//     PlcTask Inputs/GVL_iXlinker.EtherCAT_Master_EPPxxxx.Beckhoff_EPP3xxx.Beckhoff_EPP3xxxEK1122.A_0012_EPP3314_0002_0016.TC_Inputs_Channel_1.Status/Limit_2 <-> TC Inputs Channel 1/Status/Limit 2
//     PlcTask Inputs/GVL_iXlinker.EtherCAT_Master_EPPxxxx.Beckhoff_EPP3xxx.Beckhoff_EPP3xxxEK1122.A_0012_EPP3314_0002_0016.TC_Inputs_Channel_2.Status/Limit_1 <-> TC Inputs Channel 2/Status/Limit 1
//     PlcTask Inputs/GVL_iXlinker.EtherCAT_Master_EPPxxxx.Beckhoff_EPP3xxx.Beckhoff_EPP3xxxEK1122.A_0012_EPP3314_0002_0016.TC_Inputs_Channel_2.Status/Limit_2 <-> TC Inputs Channel 2/Status/Limit 2
//     PlcTask Inputs/GVL_iXlinker.EtherCAT_Master_EPPxxxx.Beckhoff_EPP3xxx.Beckhoff_EPP3xxxEK1122.A_0012_EPP3314_0002_0016.TC_Inputs_Channel_3.Status/Limit_1 <-> TC Inputs Channel 3/Status/Limit 1
//     PlcTask Inputs/GVL_iXlinker.EtherCAT_Master_EPPxxxx.Beckhoff_EPP3xxx.Beckhoff_EPP3xxxEK1122.A_0012_EPP3314_0002_0016.TC_Inputs_Channel_3.Status/Limit_2 <-> TC Inputs Channel 3/Status/Limit 2
//     PlcTask Inputs/GVL_iXlinker.EtherCAT_Master_EPPxxxx.Beckhoff_EPP3xxx.Beckhoff_EPP3xxxEK1122.A_0012_EPP3314_0002_0016.TC_Inputs_Channel_4.Status/Limit_1 <-> TC Inputs Channel 4/Status/Limit 1
//     PlcTask Inputs/GVL_iXlinker.EtherCAT_Master_EPPxxxx.Beckhoff_EPP3xxx.Beckhoff_EPP3xxxEK1122.A_0012_EPP3314_0002_0016.TC_Inputs_Channel_4.Status/Limit_2 <-> TC Inputs Channel 4/Status/Limit 2
//     PlcTask Inputs/GVL_iXlinker.EtherCAT_Master_EPPxxxx.Beckhoff_EPP3xxx.Beckhoff_EPP3xxxEK1122.A_0012_EPP3314_0002_0016.TC_Inputs_Channel_1.Status/Error <-> TC Inputs Channel 1/Status/Error
//     PlcTask Inputs/GVL_iXlinker.EtherCAT_Master_EPPxxxx.Beckhoff_EPP3xxx.Beckhoff_EPP3xxxEK1122.A_0012_EPP3314_0002_0016.TC_Inputs_Channel_2.Status/Error <-> TC Inputs Channel 2/Status/Error
//     PlcTask Inputs/GVL_iXlinker.EtherCAT_Master_EPPxxxx.Beckhoff_EPP3xxx.Beckhoff_EPP3xxxEK1122.A_0012_EPP3314_0002_0016.TC_Inputs_Channel_3.Status/Error <-> TC Inputs Channel 3/Status/Error
//     PlcTask Inputs/GVL_iXlinker.EtherCAT_Master_EPPxxxx.Beckhoff_EPP3xxx.Beckhoff_EPP3xxxEK1122.A_0012_EPP3314_0002_0016.TC_Inputs_Channel_4.Status/Error <-> TC Inputs Channel 4/Status/Error
//     PlcTask Inputs/GVL_iXlinker.EtherCAT_Master_EPPxxxx.Beckhoff_EPP3xxx.Beckhoff_EPP3xxxEK1122.A_0012_EPP3314_0002_0016.TC_Inputs_Channel_1.Status/TxPDO_State <-> TC Inputs Channel 1/Status/TxPDO State
//     PlcTask Inputs/GVL_iXlinker.EtherCAT_Master_EPPxxxx.Beckhoff_EPP3xxx.Beckhoff_EPP3xxxEK1122.A_0012_EPP3314_0002_0016.TC_Inputs_Channel_2.Status/TxPDO_State <-> TC Inputs Channel 2/Status/TxPDO State
//     PlcTask Inputs/GVL_iXlinker.EtherCAT_Master_EPPxxxx.Beckhoff_EPP3xxx.Beckhoff_EPP3xxxEK1122.A_0012_EPP3314_0002_0016.TC_Inputs_Channel_3.Status/TxPDO_State <-> TC Inputs Channel 3/Status/TxPDO State
//     PlcTask Inputs/GVL_iXlinker.EtherCAT_Master_EPPxxxx.Beckhoff_EPP3xxx.Beckhoff_EPP3xxxEK1122.A_0012_EPP3314_0002_0016.TC_Inputs_Channel_4.Status/TxPDO_State <-> TC Inputs Channel 4/Status/TxPDO State
//     PlcTask Inputs/GVL_iXlinker.EtherCAT_Master_EPPxxxx.Beckhoff_EPP3xxx.Beckhoff_EPP3xxxEK1122.A_0012_EPP3314_0002_0016.TC_Inputs_Channel_1.Status/TxPDO_Toggle <-> TC Inputs Channel 1/Status/TxPDO Toggle
//     PlcTask Inputs/GVL_iXlinker.EtherCAT_Master_EPPxxxx.Beckhoff_EPP3xxx.Beckhoff_EPP3xxxEK1122.A_0012_EPP3314_0002_0016.TC_Inputs_Channel_2.Status/TxPDO_Toggle <-> TC Inputs Channel 2/Status/TxPDO Toggle
//     PlcTask Inputs/GVL_iXlinker.EtherCAT_Master_EPPxxxx.Beckhoff_EPP3xxx.Beckhoff_EPP3xxxEK1122.A_0012_EPP3314_0002_0016.TC_Inputs_Channel_3.Status/TxPDO_Toggle <-> TC Inputs Channel 3/Status/TxPDO Toggle
//     PlcTask Inputs/GVL_iXlinker.EtherCAT_Master_EPPxxxx.Beckhoff_EPP3xxx.Beckhoff_EPP3xxxEK1122.A_0012_EPP3314_0002_0016.TC_Inputs_Channel_4.Status/TxPDO_Toggle <-> TC Inputs Channel 4/Status/TxPDO Toggle
//     PlcTask Inputs/GVL_iXlinker.EtherCAT_Master_EPPxxxx.Beckhoff_EPP3xxx.Beckhoff_EPP3xxxEK1122.A_0012_EPP3314_0002_0016.TC_Inputs_Channel_1.Value <-> TC Inputs Channel 1/Value
//     PlcTask Inputs/GVL_iXlinker.EtherCAT_Master_EPPxxxx.Beckhoff_EPP3xxx.Beckhoff_EPP3xxxEK1122.A_0012_EPP3314_0002_0016.TC_Inputs_Channel_2.Value <-> TC Inputs Channel 2/Value
//     PlcTask Inputs/GVL_iXlinker.EtherCAT_Master_EPPxxxx.Beckhoff_EPP3xxx.Beckhoff_EPP3xxxEK1122.A_0012_EPP3314_0002_0016.TC_Inputs_Channel_3.Value <-> TC Inputs Channel 3/Value
//     PlcTask Inputs/GVL_iXlinker.EtherCAT_Master_EPPxxxx.Beckhoff_EPP3xxx.Beckhoff_EPP3xxxEK1122.A_0012_EPP3314_0002_0016.TC_Inputs_Channel_4.Value <-> TC Inputs Channel 4/Value
//     PlcTask Inputs/GVL_iXlinker.EtherCAT_Master_EPPxxxx.Beckhoff_EPP3xxx.Beckhoff_EPP3xxxEK1122.A_0012_EPP3314_0002_0016.WcState.WcState <-> WcState/WcState
//     PlcTask Inputs/GVL_iXlinker.EtherCAT_Master_EPPxxxx.Beckhoff_EPP3xxx.Beckhoff_EPP3xxxEK1122.A_0012_EPP3314_0002_0016.WcState.InputToggle <-> WcState/InputToggle
//     PlcTask Inputs/GVL_iXlinker.EtherCAT_Master_EPPxxxx.Beckhoff_EPP3xxx.Beckhoff_EPP3xxxEK1122.A_0012_EPP3314_0002_0016.InfoData.AdsAddr <-> InfoData/AdsAddr
//     PlcTask Inputs/GVL_iXlinker.EtherCAT_Master_EPPxxxx.Beckhoff_EPP3xxx.Beckhoff_EPP3xxxEK1122.A_0012_EPP3314_0002_0016.InfoData.State <-> InfoData/State
//   PLC/PLC Instance <-> EtherCAT Master EPPxxxx/Beckhoff EPP3xxx/Beckhoff EPP3xxxEK1122/A_0013(EPP3314-0002-0017)
//     PlcTask Inputs/GVL_iXlinker.EtherCAT_Master_EPPxxxx.Beckhoff_EPP3xxx.Beckhoff_EPP3xxxEK1122.A_0013_EPP3314_0002_0017.TC_Inputs_Channel_1.Status/Underrange <-> TC Inputs Channel 1/Status/Underrange
//     PlcTask Inputs/GVL_iXlinker.EtherCAT_Master_EPPxxxx.Beckhoff_EPP3xxx.Beckhoff_EPP3xxxEK1122.A_0013_EPP3314_0002_0017.TC_Inputs_Channel_2.Status/Underrange <-> TC Inputs Channel 2/Status/Underrange
//     PlcTask Inputs/GVL_iXlinker.EtherCAT_Master_EPPxxxx.Beckhoff_EPP3xxx.Beckhoff_EPP3xxxEK1122.A_0013_EPP3314_0002_0017.TC_Inputs_Channel_3.Status/Underrange <-> TC Inputs Channel 3/Status/Underrange
//     PlcTask Inputs/GVL_iXlinker.EtherCAT_Master_EPPxxxx.Beckhoff_EPP3xxx.Beckhoff_EPP3xxxEK1122.A_0013_EPP3314_0002_0017.TC_Inputs_Channel_4.Status/Underrange <-> TC Inputs Channel 4/Status/Underrange
//     PlcTask Inputs/GVL_iXlinker.EtherCAT_Master_EPPxxxx.Beckhoff_EPP3xxx.Beckhoff_EPP3xxxEK1122.A_0013_EPP3314_0002_0017.TC_Inputs_Channel_1.Status/Overrange <-> TC Inputs Channel 1/Status/Overrange
//     PlcTask Inputs/GVL_iXlinker.EtherCAT_Master_EPPxxxx.Beckhoff_EPP3xxx.Beckhoff_EPP3xxxEK1122.A_0013_EPP3314_0002_0017.TC_Inputs_Channel_2.Status/Overrange <-> TC Inputs Channel 2/Status/Overrange
//     PlcTask Inputs/GVL_iXlinker.EtherCAT_Master_EPPxxxx.Beckhoff_EPP3xxx.Beckhoff_EPP3xxxEK1122.A_0013_EPP3314_0002_0017.TC_Inputs_Channel_3.Status/Overrange <-> TC Inputs Channel 3/Status/Overrange
//     PlcTask Inputs/GVL_iXlinker.EtherCAT_Master_EPPxxxx.Beckhoff_EPP3xxx.Beckhoff_EPP3xxxEK1122.A_0013_EPP3314_0002_0017.TC_Inputs_Channel_4.Status/Overrange <-> TC Inputs Channel 4/Status/Overrange
//     PlcTask Inputs/GVL_iXlinker.EtherCAT_Master_EPPxxxx.Beckhoff_EPP3xxx.Beckhoff_EPP3xxxEK1122.A_0013_EPP3314_0002_0017.TC_Inputs_Channel_1.Status/Limit_1 <-> TC Inputs Channel 1/Status/Limit 1
//     PlcTask Inputs/GVL_iXlinker.EtherCAT_Master_EPPxxxx.Beckhoff_EPP3xxx.Beckhoff_EPP3xxxEK1122.A_0013_EPP3314_0002_0017.TC_Inputs_Channel_1.Status/Limit_2 <-> TC Inputs Channel 1/Status/Limit 2
//     PlcTask Inputs/GVL_iXlinker.EtherCAT_Master_EPPxxxx.Beckhoff_EPP3xxx.Beckhoff_EPP3xxxEK1122.A_0013_EPP3314_0002_0017.TC_Inputs_Channel_2.Status/Limit_1 <-> TC Inputs Channel 2/Status/Limit 1
//     PlcTask Inputs/GVL_iXlinker.EtherCAT_Master_EPPxxxx.Beckhoff_EPP3xxx.Beckhoff_EPP3xxxEK1122.A_0013_EPP3314_0002_0017.TC_Inputs_Channel_2.Status/Limit_2 <-> TC Inputs Channel 2/Status/Limit 2
//     PlcTask Inputs/GVL_iXlinker.EtherCAT_Master_EPPxxxx.Beckhoff_EPP3xxx.Beckhoff_EPP3xxxEK1122.A_0013_EPP3314_0002_0017.TC_Inputs_Channel_3.Status/Limit_1 <-> TC Inputs Channel 3/Status/Limit 1
//     PlcTask Inputs/GVL_iXlinker.EtherCAT_Master_EPPxxxx.Beckhoff_EPP3xxx.Beckhoff_EPP3xxxEK1122.A_0013_EPP3314_0002_0017.TC_Inputs_Channel_3.Status/Limit_2 <-> TC Inputs Channel 3/Status/Limit 2
//     PlcTask Inputs/GVL_iXlinker.EtherCAT_Master_EPPxxxx.Beckhoff_EPP3xxx.Beckhoff_EPP3xxxEK1122.A_0013_EPP3314_0002_0017.TC_Inputs_Channel_4.Status/Limit_1 <-> TC Inputs Channel 4/Status/Limit 1
//     PlcTask Inputs/GVL_iXlinker.EtherCAT_Master_EPPxxxx.Beckhoff_EPP3xxx.Beckhoff_EPP3xxxEK1122.A_0013_EPP3314_0002_0017.TC_Inputs_Channel_4.Status/Limit_2 <-> TC Inputs Channel 4/Status/Limit 2
//     PlcTask Inputs/GVL_iXlinker.EtherCAT_Master_EPPxxxx.Beckhoff_EPP3xxx.Beckhoff_EPP3xxxEK1122.A_0013_EPP3314_0002_0017.TC_Inputs_Channel_1.Status/Error <-> TC Inputs Channel 1/Status/Error
//     PlcTask Inputs/GVL_iXlinker.EtherCAT_Master_EPPxxxx.Beckhoff_EPP3xxx.Beckhoff_EPP3xxxEK1122.A_0013_EPP3314_0002_0017.TC_Inputs_Channel_2.Status/Error <-> TC Inputs Channel 2/Status/Error
//     PlcTask Inputs/GVL_iXlinker.EtherCAT_Master_EPPxxxx.Beckhoff_EPP3xxx.Beckhoff_EPP3xxxEK1122.A_0013_EPP3314_0002_0017.TC_Inputs_Channel_3.Status/Error <-> TC Inputs Channel 3/Status/Error
//     PlcTask Inputs/GVL_iXlinker.EtherCAT_Master_EPPxxxx.Beckhoff_EPP3xxx.Beckhoff_EPP3xxxEK1122.A_0013_EPP3314_0002_0017.TC_Inputs_Channel_4.Status/Error <-> TC Inputs Channel 4/Status/Error
//     PlcTask Inputs/GVL_iXlinker.EtherCAT_Master_EPPxxxx.Beckhoff_EPP3xxx.Beckhoff_EPP3xxxEK1122.A_0013_EPP3314_0002_0017.TC_Inputs_Channel_1.Status/TxPDO_State <-> TC Inputs Channel 1/Status/TxPDO State
//     PlcTask Inputs/GVL_iXlinker.EtherCAT_Master_EPPxxxx.Beckhoff_EPP3xxx.Beckhoff_EPP3xxxEK1122.A_0013_EPP3314_0002_0017.TC_Inputs_Channel_2.Status/TxPDO_State <-> TC Inputs Channel 2/Status/TxPDO State
//     PlcTask Inputs/GVL_iXlinker.EtherCAT_Master_EPPxxxx.Beckhoff_EPP3xxx.Beckhoff_EPP3xxxEK1122.A_0013_EPP3314_0002_0017.TC_Inputs_Channel_3.Status/TxPDO_State <-> TC Inputs Channel 3/Status/TxPDO State
//     PlcTask Inputs/GVL_iXlinker.EtherCAT_Master_EPPxxxx.Beckhoff_EPP3xxx.Beckhoff_EPP3xxxEK1122.A_0013_EPP3314_0002_0017.TC_Inputs_Channel_4.Status/TxPDO_State <-> TC Inputs Channel 4/Status/TxPDO State
//     PlcTask Inputs/GVL_iXlinker.EtherCAT_Master_EPPxxxx.Beckhoff_EPP3xxx.Beckhoff_EPP3xxxEK1122.A_0013_EPP3314_0002_0017.TC_Inputs_Channel_1.Status/TxPDO_Toggle <-> TC Inputs Channel 1/Status/TxPDO Toggle
//     PlcTask Inputs/GVL_iXlinker.EtherCAT_Master_EPPxxxx.Beckhoff_EPP3xxx.Beckhoff_EPP3xxxEK1122.A_0013_EPP3314_0002_0017.TC_Inputs_Channel_2.Status/TxPDO_Toggle <-> TC Inputs Channel 2/Status/TxPDO Toggle
//     PlcTask Inputs/GVL_iXlinker.EtherCAT_Master_EPPxxxx.Beckhoff_EPP3xxx.Beckhoff_EPP3xxxEK1122.A_0013_EPP3314_0002_0017.TC_Inputs_Channel_3.Status/TxPDO_Toggle <-> TC Inputs Channel 3/Status/TxPDO Toggle
//     PlcTask Inputs/GVL_iXlinker.EtherCAT_Master_EPPxxxx.Beckhoff_EPP3xxx.Beckhoff_EPP3xxxEK1122.A_0013_EPP3314_0002_0017.TC_Inputs_Channel_4.Status/TxPDO_Toggle <-> TC Inputs Channel 4/Status/TxPDO Toggle
//     PlcTask Inputs/GVL_iXlinker.EtherCAT_Master_EPPxxxx.Beckhoff_EPP3xxx.Beckhoff_EPP3xxxEK1122.A_0013_EPP3314_0002_0017.TC_Inputs_Channel_1.Value <-> TC Inputs Channel 1/Value
//     PlcTask Inputs/GVL_iXlinker.EtherCAT_Master_EPPxxxx.Beckhoff_EPP3xxx.Beckhoff_EPP3xxxEK1122.A_0013_EPP3314_0002_0017.TC_Inputs_Channel_2.Value <-> TC Inputs Channel 2/Value
//     PlcTask Inputs/GVL_iXlinker.EtherCAT_Master_EPPxxxx.Beckhoff_EPP3xxx.Beckhoff_EPP3xxxEK1122.A_0013_EPP3314_0002_0017.TC_Inputs_Channel_3.Value <-> TC Inputs Channel 3/Value
//     PlcTask Inputs/GVL_iXlinker.EtherCAT_Master_EPPxxxx.Beckhoff_EPP3xxx.Beckhoff_EPP3xxxEK1122.A_0013_EPP3314_0002_0017.TC_Inputs_Channel_4.Value <-> TC Inputs Channel 4/Value
//     PlcTask Inputs/GVL_iXlinker.EtherCAT_Master_EPPxxxx.Beckhoff_EPP3xxx.Beckhoff_EPP3xxxEK1122.A_0013_EPP3314_0002_0017.WcState.WcState <-> WcState/WcState
//     PlcTask Inputs/GVL_iXlinker.EtherCAT_Master_EPPxxxx.Beckhoff_EPP3xxx.Beckhoff_EPP3xxxEK1122.A_0013_EPP3314_0002_0017.WcState.InputToggle <-> WcState/InputToggle
//     PlcTask Inputs/GVL_iXlinker.EtherCAT_Master_EPPxxxx.Beckhoff_EPP3xxx.Beckhoff_EPP3xxxEK1122.A_0013_EPP3314_0002_0017.InfoData.AdsAddr <-> InfoData/AdsAddr
//     PlcTask Inputs/GVL_iXlinker.EtherCAT_Master_EPPxxxx.Beckhoff_EPP3xxx.Beckhoff_EPP3xxxEK1122.A_0013_EPP3314_0002_0017.InfoData.State <-> InfoData/State
//   PLC/PLC Instance <-> EtherCAT Master EPPxxxx/Beckhoff EPP3xxx/Beckhoff EPP3xxxEK1122/A_0014(EPP3314-0002-0018)
//     PlcTask Inputs/GVL_iXlinker.EtherCAT_Master_EPPxxxx.Beckhoff_EPP3xxx.Beckhoff_EPP3xxxEK1122.A_0014_EPP3314_0002_0018.TC_Inputs_Channel_1.Status/Underrange <-> TC Inputs Channel 1/Status/Underrange
//     PlcTask Inputs/GVL_iXlinker.EtherCAT_Master_EPPxxxx.Beckhoff_EPP3xxx.Beckhoff_EPP3xxxEK1122.A_0014_EPP3314_0002_0018.TC_Inputs_Channel_2.Status/Underrange <-> TC Inputs Channel 2/Status/Underrange
//     PlcTask Inputs/GVL_iXlinker.EtherCAT_Master_EPPxxxx.Beckhoff_EPP3xxx.Beckhoff_EPP3xxxEK1122.A_0014_EPP3314_0002_0018.TC_Inputs_Channel_3.Status/Underrange <-> TC Inputs Channel 3/Status/Underrange
//     PlcTask Inputs/GVL_iXlinker.EtherCAT_Master_EPPxxxx.Beckhoff_EPP3xxx.Beckhoff_EPP3xxxEK1122.A_0014_EPP3314_0002_0018.TC_Inputs_Channel_4.Status/Underrange <-> TC Inputs Channel 4/Status/Underrange
//     PlcTask Inputs/GVL_iXlinker.EtherCAT_Master_EPPxxxx.Beckhoff_EPP3xxx.Beckhoff_EPP3xxxEK1122.A_0014_EPP3314_0002_0018.TC_Inputs_Channel_1.Status/Overrange <-> TC Inputs Channel 1/Status/Overrange
//     PlcTask Inputs/GVL_iXlinker.EtherCAT_Master_EPPxxxx.Beckhoff_EPP3xxx.Beckhoff_EPP3xxxEK1122.A_0014_EPP3314_0002_0018.TC_Inputs_Channel_2.Status/Overrange <-> TC Inputs Channel 2/Status/Overrange
//     PlcTask Inputs/GVL_iXlinker.EtherCAT_Master_EPPxxxx.Beckhoff_EPP3xxx.Beckhoff_EPP3xxxEK1122.A_0014_EPP3314_0002_0018.TC_Inputs_Channel_3.Status/Overrange <-> TC Inputs Channel 3/Status/Overrange
//     PlcTask Inputs/GVL_iXlinker.EtherCAT_Master_EPPxxxx.Beckhoff_EPP3xxx.Beckhoff_EPP3xxxEK1122.A_0014_EPP3314_0002_0018.TC_Inputs_Channel_4.Status/Overrange <-> TC Inputs Channel 4/Status/Overrange
//     PlcTask Inputs/GVL_iXlinker.EtherCAT_Master_EPPxxxx.Beckhoff_EPP3xxx.Beckhoff_EPP3xxxEK1122.A_0014_EPP3314_0002_0018.TC_Inputs_Channel_1.Status/Limit_1 <-> TC Inputs Channel 1/Status/Limit 1
//     PlcTask Inputs/GVL_iXlinker.EtherCAT_Master_EPPxxxx.Beckhoff_EPP3xxx.Beckhoff_EPP3xxxEK1122.A_0014_EPP3314_0002_0018.TC_Inputs_Channel_1.Status/Limit_2 <-> TC Inputs Channel 1/Status/Limit 2
//     PlcTask Inputs/GVL_iXlinker.EtherCAT_Master_EPPxxxx.Beckhoff_EPP3xxx.Beckhoff_EPP3xxxEK1122.A_0014_EPP3314_0002_0018.TC_Inputs_Channel_2.Status/Limit_1 <-> TC Inputs Channel 2/Status/Limit 1
//     PlcTask Inputs/GVL_iXlinker.EtherCAT_Master_EPPxxxx.Beckhoff_EPP3xxx.Beckhoff_EPP3xxxEK1122.A_0014_EPP3314_0002_0018.TC_Inputs_Channel_2.Status/Limit_2 <-> TC Inputs Channel 2/Status/Limit 2
//     PlcTask Inputs/GVL_iXlinker.EtherCAT_Master_EPPxxxx.Beckhoff_EPP3xxx.Beckhoff_EPP3xxxEK1122.A_0014_EPP3314_0002_0018.TC_Inputs_Channel_3.Status/Limit_1 <-> TC Inputs Channel 3/Status/Limit 1
//     PlcTask Inputs/GVL_iXlinker.EtherCAT_Master_EPPxxxx.Beckhoff_EPP3xxx.Beckhoff_EPP3xxxEK1122.A_0014_EPP3314_0002_0018.TC_Inputs_Channel_3.Status/Limit_2 <-> TC Inputs Channel 3/Status/Limit 2
//     PlcTask Inputs/GVL_iXlinker.EtherCAT_Master_EPPxxxx.Beckhoff_EPP3xxx.Beckhoff_EPP3xxxEK1122.A_0014_EPP3314_0002_0018.TC_Inputs_Channel_4.Status/Limit_1 <-> TC Inputs Channel 4/Status/Limit 1
//     PlcTask Inputs/GVL_iXlinker.EtherCAT_Master_EPPxxxx.Beckhoff_EPP3xxx.Beckhoff_EPP3xxxEK1122.A_0014_EPP3314_0002_0018.TC_Inputs_Channel_4.Status/Limit_2 <-> TC Inputs Channel 4/Status/Limit 2
//     PlcTask Inputs/GVL_iXlinker.EtherCAT_Master_EPPxxxx.Beckhoff_EPP3xxx.Beckhoff_EPP3xxxEK1122.A_0014_EPP3314_0002_0018.TC_Inputs_Channel_1.Status/Error <-> TC Inputs Channel 1/Status/Error
//     PlcTask Inputs/GVL_iXlinker.EtherCAT_Master_EPPxxxx.Beckhoff_EPP3xxx.Beckhoff_EPP3xxxEK1122.A_0014_EPP3314_0002_0018.TC_Inputs_Channel_2.Status/Error <-> TC Inputs Channel 2/Status/Error
//     PlcTask Inputs/GVL_iXlinker.EtherCAT_Master_EPPxxxx.Beckhoff_EPP3xxx.Beckhoff_EPP3xxxEK1122.A_0014_EPP3314_0002_0018.TC_Inputs_Channel_3.Status/Error <-> TC Inputs Channel 3/Status/Error
//     PlcTask Inputs/GVL_iXlinker.EtherCAT_Master_EPPxxxx.Beckhoff_EPP3xxx.Beckhoff_EPP3xxxEK1122.A_0014_EPP3314_0002_0018.TC_Inputs_Channel_4.Status/Error <-> TC Inputs Channel 4/Status/Error
//     PlcTask Inputs/GVL_iXlinker.EtherCAT_Master_EPPxxxx.Beckhoff_EPP3xxx.Beckhoff_EPP3xxxEK1122.A_0014_EPP3314_0002_0018.TC_Inputs_Channel_1.Status/TxPDO_State <-> TC Inputs Channel 1/Status/TxPDO State
//     PlcTask Inputs/GVL_iXlinker.EtherCAT_Master_EPPxxxx.Beckhoff_EPP3xxx.Beckhoff_EPP3xxxEK1122.A_0014_EPP3314_0002_0018.TC_Inputs_Channel_2.Status/TxPDO_State <-> TC Inputs Channel 2/Status/TxPDO State
//     PlcTask Inputs/GVL_iXlinker.EtherCAT_Master_EPPxxxx.Beckhoff_EPP3xxx.Beckhoff_EPP3xxxEK1122.A_0014_EPP3314_0002_0018.TC_Inputs_Channel_3.Status/TxPDO_State <-> TC Inputs Channel 3/Status/TxPDO State
//     PlcTask Inputs/GVL_iXlinker.EtherCAT_Master_EPPxxxx.Beckhoff_EPP3xxx.Beckhoff_EPP3xxxEK1122.A_0014_EPP3314_0002_0018.TC_Inputs_Channel_4.Status/TxPDO_State <-> TC Inputs Channel 4/Status/TxPDO State
//     PlcTask Inputs/GVL_iXlinker.EtherCAT_Master_EPPxxxx.Beckhoff_EPP3xxx.Beckhoff_EPP3xxxEK1122.A_0014_EPP3314_0002_0018.TC_Inputs_Channel_1.Status/TxPDO_Toggle <-> TC Inputs Channel 1/Status/TxPDO Toggle
//     PlcTask Inputs/GVL_iXlinker.EtherCAT_Master_EPPxxxx.Beckhoff_EPP3xxx.Beckhoff_EPP3xxxEK1122.A_0014_EPP3314_0002_0018.TC_Inputs_Channel_2.Status/TxPDO_Toggle <-> TC Inputs Channel 2/Status/TxPDO Toggle
//     PlcTask Inputs/GVL_iXlinker.EtherCAT_Master_EPPxxxx.Beckhoff_EPP3xxx.Beckhoff_EPP3xxxEK1122.A_0014_EPP3314_0002_0018.TC_Inputs_Channel_3.Status/TxPDO_Toggle <-> TC Inputs Channel 3/Status/TxPDO Toggle
//     PlcTask Inputs/GVL_iXlinker.EtherCAT_Master_EPPxxxx.Beckhoff_EPP3xxx.Beckhoff_EPP3xxxEK1122.A_0014_EPP3314_0002_0018.TC_Inputs_Channel_4.Status/TxPDO_Toggle <-> TC Inputs Channel 4/Status/TxPDO Toggle
//     PlcTask Inputs/GVL_iXlinker.EtherCAT_Master_EPPxxxx.Beckhoff_EPP3xxx.Beckhoff_EPP3xxxEK1122.A_0014_EPP3314_0002_0018.TC_Inputs_Channel_1.Value <-> TC Inputs Channel 1/Value
//     PlcTask Inputs/GVL_iXlinker.EtherCAT_Master_EPPxxxx.Beckhoff_EPP3xxx.Beckhoff_EPP3xxxEK1122.A_0014_EPP3314_0002_0018.TC_Inputs_Channel_2.Value <-> TC Inputs Channel 2/Value
//     PlcTask Inputs/GVL_iXlinker.EtherCAT_Master_EPPxxxx.Beckhoff_EPP3xxx.Beckhoff_EPP3xxxEK1122.A_0014_EPP3314_0002_0018.TC_Inputs_Channel_3.Value <-> TC Inputs Channel 3/Value
//     PlcTask Inputs/GVL_iXlinker.EtherCAT_Master_EPPxxxx.Beckhoff_EPP3xxx.Beckhoff_EPP3xxxEK1122.A_0014_EPP3314_0002_0018.TC_Inputs_Channel_4.Value <-> TC Inputs Channel 4/Value
//     PlcTask Inputs/GVL_iXlinker.EtherCAT_Master_EPPxxxx.Beckhoff_EPP3xxx.Beckhoff_EPP3xxxEK1122.A_0014_EPP3314_0002_0018.WcState.WcState <-> WcState/WcState
//     PlcTask Inputs/GVL_iXlinker.EtherCAT_Master_EPPxxxx.Beckhoff_EPP3xxx.Beckhoff_EPP3xxxEK1122.A_0014_EPP3314_0002_0018.WcState.InputToggle <-> WcState/InputToggle
//     PlcTask Inputs/GVL_iXlinker.EtherCAT_Master_EPPxxxx.Beckhoff_EPP3xxx.Beckhoff_EPP3xxxEK1122.A_0014_EPP3314_0002_0018.InfoData.AdsAddr <-> InfoData/AdsAddr
//     PlcTask Inputs/GVL_iXlinker.EtherCAT_Master_EPPxxxx.Beckhoff_EPP3xxx.Beckhoff_EPP3xxxEK1122.A_0014_EPP3314_0002_0018.InfoData.State <-> InfoData/State
//   PLC/PLC Instance <-> EtherCAT Master EPPxxxx/Beckhoff EPP3xxx/Beckhoff EPP3xxxEK1122/A_0015(EPP3632-0001-0016)
//     PlcTask Inputs/GVL_iXlinker.EtherCAT_Master_EPPxxxx.Beckhoff_EPP3xxx.Beckhoff_EPP3xxxEK1122.A_0015_EPP3632_0001_0016.Ch1_Status.STATUS/Underrange <-> Ch1 Status/STATUS/Underrange
//     PlcTask Inputs/GVL_iXlinker.EtherCAT_Master_EPPxxxx.Beckhoff_EPP3xxx.Beckhoff_EPP3xxxEK1122.A_0015_EPP3632_0001_0016.Ch2_Status.STATUS/Underrange <-> Ch2 Status/STATUS/Underrange
//     PlcTask Inputs/GVL_iXlinker.EtherCAT_Master_EPPxxxx.Beckhoff_EPP3xxx.Beckhoff_EPP3xxxEK1122.A_0015_EPP3632_0001_0016.Ch1_Status.STATUS/Overrange <-> Ch1 Status/STATUS/Overrange
//     PlcTask Inputs/GVL_iXlinker.EtherCAT_Master_EPPxxxx.Beckhoff_EPP3xxx.Beckhoff_EPP3xxxEK1122.A_0015_EPP3632_0001_0016.Ch2_Status.STATUS/Overrange <-> Ch2 Status/STATUS/Overrange
//     PlcTask Inputs/GVL_iXlinker.EtherCAT_Master_EPPxxxx.Beckhoff_EPP3xxx.Beckhoff_EPP3xxxEK1122.A_0015_EPP3632_0001_0016.Ch1_Status.STATUS/Limit_1 <-> Ch1 Status/STATUS/Limit 1
//     PlcTask Inputs/GVL_iXlinker.EtherCAT_Master_EPPxxxx.Beckhoff_EPP3xxx.Beckhoff_EPP3xxxEK1122.A_0015_EPP3632_0001_0016.Ch1_Status.STATUS/Limit_2 <-> Ch1 Status/STATUS/Limit 2
//     PlcTask Inputs/GVL_iXlinker.EtherCAT_Master_EPPxxxx.Beckhoff_EPP3xxx.Beckhoff_EPP3xxxEK1122.A_0015_EPP3632_0001_0016.Ch2_Status.STATUS/Limit_1 <-> Ch2 Status/STATUS/Limit 1
//     PlcTask Inputs/GVL_iXlinker.EtherCAT_Master_EPPxxxx.Beckhoff_EPP3xxx.Beckhoff_EPP3xxxEK1122.A_0015_EPP3632_0001_0016.Ch2_Status.STATUS/Limit_2 <-> Ch2 Status/STATUS/Limit 2
//     PlcTask Inputs/GVL_iXlinker.EtherCAT_Master_EPPxxxx.Beckhoff_EPP3xxx.Beckhoff_EPP3xxxEK1122.A_0015_EPP3632_0001_0016.Ch1_Status.STATUS/Error <-> Ch1 Status/STATUS/Error
//     PlcTask Inputs/GVL_iXlinker.EtherCAT_Master_EPPxxxx.Beckhoff_EPP3xxx.Beckhoff_EPP3xxxEK1122.A_0015_EPP3632_0001_0016.Ch2_Status.STATUS/Error <-> Ch2 Status/STATUS/Error
//     PlcTask Inputs/GVL_iXlinker.EtherCAT_Master_EPPxxxx.Beckhoff_EPP3xxx.Beckhoff_EPP3xxxEK1122.A_0015_EPP3632_0001_0016.Ch1_Status.STATUS/Sync_error <-> Ch1 Status/STATUS/Sync error
//     PlcTask Inputs/GVL_iXlinker.EtherCAT_Master_EPPxxxx.Beckhoff_EPP3xxx.Beckhoff_EPP3xxxEK1122.A_0015_EPP3632_0001_0016.Ch2_Status.STATUS/Sync_error <-> Ch2 Status/STATUS/Sync error
//     PlcTask Inputs/GVL_iXlinker.EtherCAT_Master_EPPxxxx.Beckhoff_EPP3xxx.Beckhoff_EPP3xxxEK1122.A_0015_EPP3632_0001_0016.Ch1_Status.STATUS/TxPDO_State <-> Ch1 Status/STATUS/TxPDO State
//     PlcTask Inputs/GVL_iXlinker.EtherCAT_Master_EPPxxxx.Beckhoff_EPP3xxx.Beckhoff_EPP3xxxEK1122.A_0015_EPP3632_0001_0016.Ch2_Status.STATUS/TxPDO_State <-> Ch2 Status/STATUS/TxPDO State
//     PlcTask Inputs/GVL_iXlinker.EtherCAT_Master_EPPxxxx.Beckhoff_EPP3xxx.Beckhoff_EPP3xxxEK1122.A_0015_EPP3632_0001_0016.Ch1_Status.STATUS/TxPDO_Toggle <-> Ch1 Status/STATUS/TxPDO Toggle
//     PlcTask Inputs/GVL_iXlinker.EtherCAT_Master_EPPxxxx.Beckhoff_EPP3xxx.Beckhoff_EPP3xxxEK1122.A_0015_EPP3632_0001_0016.Ch2_Status.STATUS/TxPDO_Toggle <-> Ch2 Status/STATUS/TxPDO Toggle
//     PlcTask Inputs/GVL_iXlinker.EtherCAT_Master_EPPxxxx.Beckhoff_EPP3xxx.Beckhoff_EPP3xxxEK1122.A_0015_EPP3632_0001_0016.Ch1_Sample_0.Ch1_Value <-> Ch1 Sample 0/Ch1 Value
//     PlcTask Inputs/GVL_iXlinker.EtherCAT_Master_EPPxxxx.Beckhoff_EPP3xxx.Beckhoff_EPP3xxxEK1122.A_0015_EPP3632_0001_0016.Ch1_Sample_1.Ch1_Value <-> Ch1 Sample 1/Ch1 Value
//     PlcTask Inputs/GVL_iXlinker.EtherCAT_Master_EPPxxxx.Beckhoff_EPP3xxx.Beckhoff_EPP3xxxEK1122.A_0015_EPP3632_0001_0016.Ch1_Sample_2.Ch1_Value <-> Ch1 Sample 2/Ch1 Value
//     PlcTask Inputs/GVL_iXlinker.EtherCAT_Master_EPPxxxx.Beckhoff_EPP3xxx.Beckhoff_EPP3xxxEK1122.A_0015_EPP3632_0001_0016.Ch1_Sample_3.Ch1_Value <-> Ch1 Sample 3/Ch1 Value
//     PlcTask Inputs/GVL_iXlinker.EtherCAT_Master_EPPxxxx.Beckhoff_EPP3xxx.Beckhoff_EPP3xxxEK1122.A_0015_EPP3632_0001_0016.Ch1_Sample_4.Ch1_Value <-> Ch1 Sample 4/Ch1 Value
//     PlcTask Inputs/GVL_iXlinker.EtherCAT_Master_EPPxxxx.Beckhoff_EPP3xxx.Beckhoff_EPP3xxxEK1122.A_0015_EPP3632_0001_0016.Ch1_Sample_5.Ch1_Value <-> Ch1 Sample 5/Ch1 Value
//     PlcTask Inputs/GVL_iXlinker.EtherCAT_Master_EPPxxxx.Beckhoff_EPP3xxx.Beckhoff_EPP3xxxEK1122.A_0015_EPP3632_0001_0016.Ch1_Sample_6.Ch1_Value <-> Ch1 Sample 6/Ch1 Value
//     PlcTask Inputs/GVL_iXlinker.EtherCAT_Master_EPPxxxx.Beckhoff_EPP3xxx.Beckhoff_EPP3xxxEK1122.A_0015_EPP3632_0001_0016.Ch1_Sample_7.Ch1_Value <-> Ch1 Sample 7/Ch1 Value
//     PlcTask Inputs/GVL_iXlinker.EtherCAT_Master_EPPxxxx.Beckhoff_EPP3xxx.Beckhoff_EPP3xxxEK1122.A_0015_EPP3632_0001_0016.Ch1_Sample_8.Ch1_Value <-> Ch1 Sample 8/Ch1 Value
//     PlcTask Inputs/GVL_iXlinker.EtherCAT_Master_EPPxxxx.Beckhoff_EPP3xxx.Beckhoff_EPP3xxxEK1122.A_0015_EPP3632_0001_0016.Ch1_Sample_9.Ch1_Value <-> Ch1 Sample 9/Ch1 Value
//     PlcTask Inputs/GVL_iXlinker.EtherCAT_Master_EPPxxxx.Beckhoff_EPP3xxx.Beckhoff_EPP3xxxEK1122.A_0015_EPP3632_0001_0016.Ch2_Sample_0.Ch2_Value <-> Ch2 Sample 0/Ch2 Value
//     PlcTask Inputs/GVL_iXlinker.EtherCAT_Master_EPPxxxx.Beckhoff_EPP3xxx.Beckhoff_EPP3xxxEK1122.A_0015_EPP3632_0001_0016.Ch2_Sample_1.Ch2_Value <-> Ch2 Sample 1/Ch2 Value
//     PlcTask Inputs/GVL_iXlinker.EtherCAT_Master_EPPxxxx.Beckhoff_EPP3xxx.Beckhoff_EPP3xxxEK1122.A_0015_EPP3632_0001_0016.Ch2_Sample_2.Ch2_Value <-> Ch2 Sample 2/Ch2 Value
//     PlcTask Inputs/GVL_iXlinker.EtherCAT_Master_EPPxxxx.Beckhoff_EPP3xxx.Beckhoff_EPP3xxxEK1122.A_0015_EPP3632_0001_0016.Ch2_Sample_3.Ch2_Value <-> Ch2 Sample 3/Ch2 Value
//     PlcTask Inputs/GVL_iXlinker.EtherCAT_Master_EPPxxxx.Beckhoff_EPP3xxx.Beckhoff_EPP3xxxEK1122.A_0015_EPP3632_0001_0016.Ch2_Sample_4.Ch2_Value <-> Ch2 Sample 4/Ch2 Value
//     PlcTask Inputs/GVL_iXlinker.EtherCAT_Master_EPPxxxx.Beckhoff_EPP3xxx.Beckhoff_EPP3xxxEK1122.A_0015_EPP3632_0001_0016.Ch2_Sample_5.Ch2_Value <-> Ch2 Sample 5/Ch2 Value
//     PlcTask Inputs/GVL_iXlinker.EtherCAT_Master_EPPxxxx.Beckhoff_EPP3xxx.Beckhoff_EPP3xxxEK1122.A_0015_EPP3632_0001_0016.Ch2_Sample_6.Ch2_Value <-> Ch2 Sample 6/Ch2 Value
//     PlcTask Inputs/GVL_iXlinker.EtherCAT_Master_EPPxxxx.Beckhoff_EPP3xxx.Beckhoff_EPP3xxxEK1122.A_0015_EPP3632_0001_0016.Ch2_Sample_7.Ch2_Value <-> Ch2 Sample 7/Ch2 Value
//     PlcTask Inputs/GVL_iXlinker.EtherCAT_Master_EPPxxxx.Beckhoff_EPP3xxx.Beckhoff_EPP3xxxEK1122.A_0015_EPP3632_0001_0016.Ch2_Sample_8.Ch2_Value <-> Ch2 Sample 8/Ch2 Value
//     PlcTask Inputs/GVL_iXlinker.EtherCAT_Master_EPPxxxx.Beckhoff_EPP3xxx.Beckhoff_EPP3xxxEK1122.A_0015_EPP3632_0001_0016.Ch2_Sample_9.Ch2_Value <-> Ch2 Sample 9/Ch2 Value
//     PlcTask Inputs/GVL_iXlinker.EtherCAT_Master_EPPxxxx.Beckhoff_EPP3xxx.Beckhoff_EPP3xxxEK1122.A_0015_EPP3632_0001_0016.NextSync1Time.StartTimeNextLatch <-> NextSync1Time/StartTimeNextLatch
//     PlcTask Inputs/GVL_iXlinker.EtherCAT_Master_EPPxxxx.Beckhoff_EPP3xxx.Beckhoff_EPP3xxxEK1122.A_0015_EPP3632_0001_0016.Sample_Count.Sample_Count <-> Sample Count/Sample Count
//     PlcTask Inputs/GVL_iXlinker.EtherCAT_Master_EPPxxxx.Beckhoff_EPP3xxx.Beckhoff_EPP3xxxEK1122.A_0015_EPP3632_0001_0016.WcState.WcState <-> WcState/WcState
//     PlcTask Inputs/GVL_iXlinker.EtherCAT_Master_EPPxxxx.Beckhoff_EPP3xxx.Beckhoff_EPP3xxxEK1122.A_0015_EPP3632_0001_0016.WcState.InputToggle <-> WcState/InputToggle
//     PlcTask Inputs/GVL_iXlinker.EtherCAT_Master_EPPxxxx.Beckhoff_EPP3xxx.Beckhoff_EPP3xxxEK1122.A_0015_EPP3632_0001_0016.InfoData.AdsAddr <-> InfoData/AdsAddr
//     PlcTask Inputs/GVL_iXlinker.EtherCAT_Master_EPPxxxx.Beckhoff_EPP3xxx.Beckhoff_EPP3xxxEK1122.A_0015_EPP3632_0001_0016.InfoData.DcOutputShift <-> InfoData/DcOutputShift
//     PlcTask Inputs/GVL_iXlinker.EtherCAT_Master_EPPxxxx.Beckhoff_EPP3xxx.Beckhoff_EPP3xxxEK1122.A_0015_EPP3632_0001_0016.InfoData.DcInputShift <-> InfoData/DcInputShift
//     PlcTask Inputs/GVL_iXlinker.EtherCAT_Master_EPPxxxx.Beckhoff_EPP3xxx.Beckhoff_EPP3xxxEK1122.A_0015_EPP3632_0001_0016.InfoData.State <-> InfoData/State
//   PLC/PLC Instance <-> EtherCAT Master EPPxxxx/Beckhoff EPP3xxx/Beckhoff EPP3xxxEK1122/A_0016(EPP3632-0001-0017)
//     PlcTask Inputs/GVL_iXlinker.EtherCAT_Master_EPPxxxx.Beckhoff_EPP3xxx.Beckhoff_EPP3xxxEK1122.A_0016_EPP3632_0001_0017.Ch1_Status.STATUS/Underrange <-> Ch1 Status/STATUS/Underrange
//     PlcTask Inputs/GVL_iXlinker.EtherCAT_Master_EPPxxxx.Beckhoff_EPP3xxx.Beckhoff_EPP3xxxEK1122.A_0016_EPP3632_0001_0017.Ch2_Status.STATUS/Underrange <-> Ch2 Status/STATUS/Underrange
//     PlcTask Inputs/GVL_iXlinker.EtherCAT_Master_EPPxxxx.Beckhoff_EPP3xxx.Beckhoff_EPP3xxxEK1122.A_0016_EPP3632_0001_0017.Ch1_Status.STATUS/Overrange <-> Ch1 Status/STATUS/Overrange
//     PlcTask Inputs/GVL_iXlinker.EtherCAT_Master_EPPxxxx.Beckhoff_EPP3xxx.Beckhoff_EPP3xxxEK1122.A_0016_EPP3632_0001_0017.Ch2_Status.STATUS/Overrange <-> Ch2 Status/STATUS/Overrange
//     PlcTask Inputs/GVL_iXlinker.EtherCAT_Master_EPPxxxx.Beckhoff_EPP3xxx.Beckhoff_EPP3xxxEK1122.A_0016_EPP3632_0001_0017.Ch1_Status.STATUS/Limit_1 <-> Ch1 Status/STATUS/Limit 1
//     PlcTask Inputs/GVL_iXlinker.EtherCAT_Master_EPPxxxx.Beckhoff_EPP3xxx.Beckhoff_EPP3xxxEK1122.A_0016_EPP3632_0001_0017.Ch1_Status.STATUS/Limit_2 <-> Ch1 Status/STATUS/Limit 2
//     PlcTask Inputs/GVL_iXlinker.EtherCAT_Master_EPPxxxx.Beckhoff_EPP3xxx.Beckhoff_EPP3xxxEK1122.A_0016_EPP3632_0001_0017.Ch2_Status.STATUS/Limit_1 <-> Ch2 Status/STATUS/Limit 1
//     PlcTask Inputs/GVL_iXlinker.EtherCAT_Master_EPPxxxx.Beckhoff_EPP3xxx.Beckhoff_EPP3xxxEK1122.A_0016_EPP3632_0001_0017.Ch2_Status.STATUS/Limit_2 <-> Ch2 Status/STATUS/Limit 2
//     PlcTask Inputs/GVL_iXlinker.EtherCAT_Master_EPPxxxx.Beckhoff_EPP3xxx.Beckhoff_EPP3xxxEK1122.A_0016_EPP3632_0001_0017.Ch1_Status.STATUS/Error <-> Ch1 Status/STATUS/Error
//     PlcTask Inputs/GVL_iXlinker.EtherCAT_Master_EPPxxxx.Beckhoff_EPP3xxx.Beckhoff_EPP3xxxEK1122.A_0016_EPP3632_0001_0017.Ch2_Status.STATUS/Error <-> Ch2 Status/STATUS/Error
//     PlcTask Inputs/GVL_iXlinker.EtherCAT_Master_EPPxxxx.Beckhoff_EPP3xxx.Beckhoff_EPP3xxxEK1122.A_0016_EPP3632_0001_0017.Ch1_Status.STATUS/Sync_error <-> Ch1 Status/STATUS/Sync error
//     PlcTask Inputs/GVL_iXlinker.EtherCAT_Master_EPPxxxx.Beckhoff_EPP3xxx.Beckhoff_EPP3xxxEK1122.A_0016_EPP3632_0001_0017.Ch2_Status.STATUS/Sync_error <-> Ch2 Status/STATUS/Sync error
//     PlcTask Inputs/GVL_iXlinker.EtherCAT_Master_EPPxxxx.Beckhoff_EPP3xxx.Beckhoff_EPP3xxxEK1122.A_0016_EPP3632_0001_0017.Ch1_Status.STATUS/TxPDO_State <-> Ch1 Status/STATUS/TxPDO State
//     PlcTask Inputs/GVL_iXlinker.EtherCAT_Master_EPPxxxx.Beckhoff_EPP3xxx.Beckhoff_EPP3xxxEK1122.A_0016_EPP3632_0001_0017.Ch2_Status.STATUS/TxPDO_State <-> Ch2 Status/STATUS/TxPDO State
//     PlcTask Inputs/GVL_iXlinker.EtherCAT_Master_EPPxxxx.Beckhoff_EPP3xxx.Beckhoff_EPP3xxxEK1122.A_0016_EPP3632_0001_0017.Ch1_Status.STATUS/TxPDO_Toggle <-> Ch1 Status/STATUS/TxPDO Toggle
//     PlcTask Inputs/GVL_iXlinker.EtherCAT_Master_EPPxxxx.Beckhoff_EPP3xxx.Beckhoff_EPP3xxxEK1122.A_0016_EPP3632_0001_0017.Ch2_Status.STATUS/TxPDO_Toggle <-> Ch2 Status/STATUS/TxPDO Toggle
//     PlcTask Inputs/GVL_iXlinker.EtherCAT_Master_EPPxxxx.Beckhoff_EPP3xxx.Beckhoff_EPP3xxxEK1122.A_0016_EPP3632_0001_0017.Ch1_Sample_0.Ch1_Value <-> Ch1 Sample 0/Ch1 Value
//     PlcTask Inputs/GVL_iXlinker.EtherCAT_Master_EPPxxxx.Beckhoff_EPP3xxx.Beckhoff_EPP3xxxEK1122.A_0016_EPP3632_0001_0017.Ch1_Sample_1.Ch1_Value <-> Ch1 Sample 1/Ch1 Value
//     PlcTask Inputs/GVL_iXlinker.EtherCAT_Master_EPPxxxx.Beckhoff_EPP3xxx.Beckhoff_EPP3xxxEK1122.A_0016_EPP3632_0001_0017.Ch1_Sample_2.Ch1_Value <-> Ch1 Sample 2/Ch1 Value
//     PlcTask Inputs/GVL_iXlinker.EtherCAT_Master_EPPxxxx.Beckhoff_EPP3xxx.Beckhoff_EPP3xxxEK1122.A_0016_EPP3632_0001_0017.Ch1_Sample_3.Ch1_Value <-> Ch1 Sample 3/Ch1 Value
//     PlcTask Inputs/GVL_iXlinker.EtherCAT_Master_EPPxxxx.Beckhoff_EPP3xxx.Beckhoff_EPP3xxxEK1122.A_0016_EPP3632_0001_0017.Ch1_Sample_4.Ch1_Value <-> Ch1 Sample 4/Ch1 Value
//     PlcTask Inputs/GVL_iXlinker.EtherCAT_Master_EPPxxxx.Beckhoff_EPP3xxx.Beckhoff_EPP3xxxEK1122.A_0016_EPP3632_0001_0017.Ch1_Sample_5.Ch1_Value <-> Ch1 Sample 5/Ch1 Value
//     PlcTask Inputs/GVL_iXlinker.EtherCAT_Master_EPPxxxx.Beckhoff_EPP3xxx.Beckhoff_EPP3xxxEK1122.A_0016_EPP3632_0001_0017.Ch1_Sample_6.Ch1_Value <-> Ch1 Sample 6/Ch1 Value
//     PlcTask Inputs/GVL_iXlinker.EtherCAT_Master_EPPxxxx.Beckhoff_EPP3xxx.Beckhoff_EPP3xxxEK1122.A_0016_EPP3632_0001_0017.Ch1_Sample_7.Ch1_Value <-> Ch1 Sample 7/Ch1 Value
//     PlcTask Inputs/GVL_iXlinker.EtherCAT_Master_EPPxxxx.Beckhoff_EPP3xxx.Beckhoff_EPP3xxxEK1122.A_0016_EPP3632_0001_0017.Ch1_Sample_8.Ch1_Value <-> Ch1 Sample 8/Ch1 Value
//     PlcTask Inputs/GVL_iXlinker.EtherCAT_Master_EPPxxxx.Beckhoff_EPP3xxx.Beckhoff_EPP3xxxEK1122.A_0016_EPP3632_0001_0017.Ch1_Sample_9.Ch1_Value <-> Ch1 Sample 9/Ch1 Value
//     PlcTask Inputs/GVL_iXlinker.EtherCAT_Master_EPPxxxx.Beckhoff_EPP3xxx.Beckhoff_EPP3xxxEK1122.A_0016_EPP3632_0001_0017.Ch2_Sample_0.Ch2_Value <-> Ch2 Sample 0/Ch2 Value
//     PlcTask Inputs/GVL_iXlinker.EtherCAT_Master_EPPxxxx.Beckhoff_EPP3xxx.Beckhoff_EPP3xxxEK1122.A_0016_EPP3632_0001_0017.Ch2_Sample_1.Ch2_Value <-> Ch2 Sample 1/Ch2 Value
//     PlcTask Inputs/GVL_iXlinker.EtherCAT_Master_EPPxxxx.Beckhoff_EPP3xxx.Beckhoff_EPP3xxxEK1122.A_0016_EPP3632_0001_0017.Ch2_Sample_2.Ch2_Value <-> Ch2 Sample 2/Ch2 Value
//     PlcTask Inputs/GVL_iXlinker.EtherCAT_Master_EPPxxxx.Beckhoff_EPP3xxx.Beckhoff_EPP3xxxEK1122.A_0016_EPP3632_0001_0017.Ch2_Sample_3.Ch2_Value <-> Ch2 Sample 3/Ch2 Value
//     PlcTask Inputs/GVL_iXlinker.EtherCAT_Master_EPPxxxx.Beckhoff_EPP3xxx.Beckhoff_EPP3xxxEK1122.A_0016_EPP3632_0001_0017.Ch2_Sample_4.Ch2_Value <-> Ch2 Sample 4/Ch2 Value
//     PlcTask Inputs/GVL_iXlinker.EtherCAT_Master_EPPxxxx.Beckhoff_EPP3xxx.Beckhoff_EPP3xxxEK1122.A_0016_EPP3632_0001_0017.Ch2_Sample_5.Ch2_Value <-> Ch2 Sample 5/Ch2 Value
//     PlcTask Inputs/GVL_iXlinker.EtherCAT_Master_EPPxxxx.Beckhoff_EPP3xxx.Beckhoff_EPP3xxxEK1122.A_0016_EPP3632_0001_0017.Ch2_Sample_6.Ch2_Value <-> Ch2 Sample 6/Ch2 Value
//     PlcTask Inputs/GVL_iXlinker.EtherCAT_Master_EPPxxxx.Beckhoff_EPP3xxx.Beckhoff_EPP3xxxEK1122.A_0016_EPP3632_0001_0017.Ch2_Sample_7.Ch2_Value <-> Ch2 Sample 7/Ch2 Value
//     PlcTask Inputs/GVL_iXlinker.EtherCAT_Master_EPPxxxx.Beckhoff_EPP3xxx.Beckhoff_EPP3xxxEK1122.A_0016_EPP3632_0001_0017.Ch2_Sample_8.Ch2_Value <-> Ch2 Sample 8/Ch2 Value
//     PlcTask Inputs/GVL_iXlinker.EtherCAT_Master_EPPxxxx.Beckhoff_EPP3xxx.Beckhoff_EPP3xxxEK1122.A_0016_EPP3632_0001_0017.Ch2_Sample_9.Ch2_Value <-> Ch2 Sample 9/Ch2 Value
//     PlcTask Inputs/GVL_iXlinker.EtherCAT_Master_EPPxxxx.Beckhoff_EPP3xxx.Beckhoff_EPP3xxxEK1122.A_0016_EPP3632_0001_0017.NextSync1Time.StartTimeNextLatch <-> NextSync1Time/StartTimeNextLatch
//     PlcTask Inputs/GVL_iXlinker.EtherCAT_Master_EPPxxxx.Beckhoff_EPP3xxx.Beckhoff_EPP3xxxEK1122.A_0016_EPP3632_0001_0017.Sample_Count.Sample_Count <-> Sample Count/Sample Count
//     PlcTask Inputs/GVL_iXlinker.EtherCAT_Master_EPPxxxx.Beckhoff_EPP3xxx.Beckhoff_EPP3xxxEK1122.A_0016_EPP3632_0001_0017.WcState.WcState <-> WcState/WcState
//     PlcTask Inputs/GVL_iXlinker.EtherCAT_Master_EPPxxxx.Beckhoff_EPP3xxx.Beckhoff_EPP3xxxEK1122.A_0016_EPP3632_0001_0017.WcState.InputToggle <-> WcState/InputToggle
//     PlcTask Inputs/GVL_iXlinker.EtherCAT_Master_EPPxxxx.Beckhoff_EPP3xxx.Beckhoff_EPP3xxxEK1122.A_0016_EPP3632_0001_0017.InfoData.AdsAddr <-> InfoData/AdsAddr
//     PlcTask Inputs/GVL_iXlinker.EtherCAT_Master_EPPxxxx.Beckhoff_EPP3xxx.Beckhoff_EPP3xxxEK1122.A_0016_EPP3632_0001_0017.InfoData.DcOutputShift <-> InfoData/DcOutputShift
//     PlcTask Inputs/GVL_iXlinker.EtherCAT_Master_EPPxxxx.Beckhoff_EPP3xxx.Beckhoff_EPP3xxxEK1122.A_0016_EPP3632_0001_0017.InfoData.DcInputShift <-> InfoData/DcInputShift
//     PlcTask Inputs/GVL_iXlinker.EtherCAT_Master_EPPxxxx.Beckhoff_EPP3xxx.Beckhoff_EPP3xxxEK1122.A_0016_EPP3632_0001_0017.InfoData.State <-> InfoData/State
//   PLC/PLC Instance <-> EtherCAT Master EPPxxxx/Beckhoff EPP3xxx/Beckhoff EPP3xxxEK1122/A_0017(EPP3744-0041-0016)
//     PlcTask Inputs/GVL_iXlinker.EtherCAT_Master_EPPxxxx.Beckhoff_EPP3xxx.Beckhoff_EPP3xxxEK1122.A_0017_EPP3744_0041_0016.DIG_Inputs.Input[0] <-> DIG Inputs/Input 1
//     PlcTask Inputs/GVL_iXlinker.EtherCAT_Master_EPPxxxx.Beckhoff_EPP3xxx.Beckhoff_EPP3xxxEK1122.A_0017_EPP3744_0041_0016.DIG_Inputs.Input[1] <-> DIG Inputs/Input 2
//     PlcTask Inputs/GVL_iXlinker.EtherCAT_Master_EPPxxxx.Beckhoff_EPP3xxx.Beckhoff_EPP3xxxEK1122.A_0017_EPP3744_0041_0016.DIG_Inputs.Input[2] <-> DIG Inputs/Input 3
//     PlcTask Inputs/GVL_iXlinker.EtherCAT_Master_EPPxxxx.Beckhoff_EPP3xxx.Beckhoff_EPP3xxxEK1122.A_0017_EPP3744_0041_0016.DIG_Inputs.Input[3] <-> DIG Inputs/Input 4
//     PlcTask Inputs/GVL_iXlinker.EtherCAT_Master_EPPxxxx.Beckhoff_EPP3xxx.Beckhoff_EPP3xxxEK1122.A_0017_EPP3744_0041_0016.DIG_Inputs.Input[4] <-> DIG Inputs/Input 5
//     PlcTask Inputs/GVL_iXlinker.EtherCAT_Master_EPPxxxx.Beckhoff_EPP3xxx.Beckhoff_EPP3xxxEK1122.A_0017_EPP3744_0041_0016.DIG_Inputs.Input[5] <-> DIG Inputs/Input 6
//     PlcTask Inputs/GVL_iXlinker.EtherCAT_Master_EPPxxxx.Beckhoff_EPP3xxx.Beckhoff_EPP3xxxEK1122.A_0017_EPP3744_0041_0016.AI_Inputs_Channel_1.Status/Underrange <-> AI Inputs Channel 1/Status/Underrange
//     PlcTask Inputs/GVL_iXlinker.EtherCAT_Master_EPPxxxx.Beckhoff_EPP3xxx.Beckhoff_EPP3xxxEK1122.A_0017_EPP3744_0041_0016.AI_Inputs_Channel_2.Status/Underrange <-> AI Inputs Channel 2/Status/Underrange
//     PlcTask Inputs/GVL_iXlinker.EtherCAT_Master_EPPxxxx.Beckhoff_EPP3xxx.Beckhoff_EPP3xxxEK1122.A_0017_EPP3744_0041_0016.AI_Inputs_Channel_3.Status/Underrange <-> AI Inputs Channel 3/Status/Underrange
//     PlcTask Inputs/GVL_iXlinker.EtherCAT_Master_EPPxxxx.Beckhoff_EPP3xxx.Beckhoff_EPP3xxxEK1122.A_0017_EPP3744_0041_0016.AI_Inputs_Channel_4.Status/Underrange <-> AI Inputs Channel 4/Status/Underrange
//     PlcTask Inputs/GVL_iXlinker.EtherCAT_Master_EPPxxxx.Beckhoff_EPP3xxx.Beckhoff_EPP3xxxEK1122.A_0017_EPP3744_0041_0016.AI_Inputs_Channel_1.Status/Overrange <-> AI Inputs Channel 1/Status/Overrange
//     PlcTask Inputs/GVL_iXlinker.EtherCAT_Master_EPPxxxx.Beckhoff_EPP3xxx.Beckhoff_EPP3xxxEK1122.A_0017_EPP3744_0041_0016.AI_Inputs_Channel_2.Status/Overrange <-> AI Inputs Channel 2/Status/Overrange
//     PlcTask Inputs/GVL_iXlinker.EtherCAT_Master_EPPxxxx.Beckhoff_EPP3xxx.Beckhoff_EPP3xxxEK1122.A_0017_EPP3744_0041_0016.AI_Inputs_Channel_3.Status/Overrange <-> AI Inputs Channel 3/Status/Overrange
//     PlcTask Inputs/GVL_iXlinker.EtherCAT_Master_EPPxxxx.Beckhoff_EPP3xxx.Beckhoff_EPP3xxxEK1122.A_0017_EPP3744_0041_0016.AI_Inputs_Channel_4.Status/Overrange <-> AI Inputs Channel 4/Status/Overrange
//     PlcTask Inputs/GVL_iXlinker.EtherCAT_Master_EPPxxxx.Beckhoff_EPP3xxx.Beckhoff_EPP3xxxEK1122.A_0017_EPP3744_0041_0016.AI_Inputs_Channel_1.Status/Limit_1 <-> AI Inputs Channel 1/Status/Limit 1
//     PlcTask Inputs/GVL_iXlinker.EtherCAT_Master_EPPxxxx.Beckhoff_EPP3xxx.Beckhoff_EPP3xxxEK1122.A_0017_EPP3744_0041_0016.AI_Inputs_Channel_1.Status/Limit_2 <-> AI Inputs Channel 1/Status/Limit 2
//     PlcTask Inputs/GVL_iXlinker.EtherCAT_Master_EPPxxxx.Beckhoff_EPP3xxx.Beckhoff_EPP3xxxEK1122.A_0017_EPP3744_0041_0016.AI_Inputs_Channel_2.Status/Limit_1 <-> AI Inputs Channel 2/Status/Limit 1
//     PlcTask Inputs/GVL_iXlinker.EtherCAT_Master_EPPxxxx.Beckhoff_EPP3xxx.Beckhoff_EPP3xxxEK1122.A_0017_EPP3744_0041_0016.AI_Inputs_Channel_2.Status/Limit_2 <-> AI Inputs Channel 2/Status/Limit 2
//     PlcTask Inputs/GVL_iXlinker.EtherCAT_Master_EPPxxxx.Beckhoff_EPP3xxx.Beckhoff_EPP3xxxEK1122.A_0017_EPP3744_0041_0016.AI_Inputs_Channel_3.Status/Limit_1 <-> AI Inputs Channel 3/Status/Limit 1
//     PlcTask Inputs/GVL_iXlinker.EtherCAT_Master_EPPxxxx.Beckhoff_EPP3xxx.Beckhoff_EPP3xxxEK1122.A_0017_EPP3744_0041_0016.AI_Inputs_Channel_3.Status/Limit_2 <-> AI Inputs Channel 3/Status/Limit 2
//     PlcTask Inputs/GVL_iXlinker.EtherCAT_Master_EPPxxxx.Beckhoff_EPP3xxx.Beckhoff_EPP3xxxEK1122.A_0017_EPP3744_0041_0016.AI_Inputs_Channel_4.Status/Limit_1 <-> AI Inputs Channel 4/Status/Limit 1
//     PlcTask Inputs/GVL_iXlinker.EtherCAT_Master_EPPxxxx.Beckhoff_EPP3xxx.Beckhoff_EPP3xxxEK1122.A_0017_EPP3744_0041_0016.AI_Inputs_Channel_4.Status/Limit_2 <-> AI Inputs Channel 4/Status/Limit 2
//     PlcTask Inputs/GVL_iXlinker.EtherCAT_Master_EPPxxxx.Beckhoff_EPP3xxx.Beckhoff_EPP3xxxEK1122.A_0017_EPP3744_0041_0016.AI_Inputs_Channel_1.Status/Error <-> AI Inputs Channel 1/Status/Error
//     PlcTask Inputs/GVL_iXlinker.EtherCAT_Master_EPPxxxx.Beckhoff_EPP3xxx.Beckhoff_EPP3xxxEK1122.A_0017_EPP3744_0041_0016.AI_Inputs_Channel_2.Status/Error <-> AI Inputs Channel 2/Status/Error
//     PlcTask Inputs/GVL_iXlinker.EtherCAT_Master_EPPxxxx.Beckhoff_EPP3xxx.Beckhoff_EPP3xxxEK1122.A_0017_EPP3744_0041_0016.AI_Inputs_Channel_3.Status/Error <-> AI Inputs Channel 3/Status/Error
//     PlcTask Inputs/GVL_iXlinker.EtherCAT_Master_EPPxxxx.Beckhoff_EPP3xxx.Beckhoff_EPP3xxxEK1122.A_0017_EPP3744_0041_0016.AI_Inputs_Channel_4.Status/Error <-> AI Inputs Channel 4/Status/Error
//     PlcTask Inputs/GVL_iXlinker.EtherCAT_Master_EPPxxxx.Beckhoff_EPP3xxx.Beckhoff_EPP3xxxEK1122.A_0017_EPP3744_0041_0016.AI_Inputs_Channel_1.Status/TxPDO_State <-> AI Inputs Channel 1/Status/TxPDO State
//     PlcTask Inputs/GVL_iXlinker.EtherCAT_Master_EPPxxxx.Beckhoff_EPP3xxx.Beckhoff_EPP3xxxEK1122.A_0017_EPP3744_0041_0016.AI_Inputs_Channel_2.Status/TxPDO_State <-> AI Inputs Channel 2/Status/TxPDO State
//     PlcTask Inputs/GVL_iXlinker.EtherCAT_Master_EPPxxxx.Beckhoff_EPP3xxx.Beckhoff_EPP3xxxEK1122.A_0017_EPP3744_0041_0016.AI_Inputs_Channel_3.Status/TxPDO_State <-> AI Inputs Channel 3/Status/TxPDO State
//     PlcTask Inputs/GVL_iXlinker.EtherCAT_Master_EPPxxxx.Beckhoff_EPP3xxx.Beckhoff_EPP3xxxEK1122.A_0017_EPP3744_0041_0016.AI_Inputs_Channel_4.Status/TxPDO_State <-> AI Inputs Channel 4/Status/TxPDO State
//     PlcTask Inputs/GVL_iXlinker.EtherCAT_Master_EPPxxxx.Beckhoff_EPP3xxx.Beckhoff_EPP3xxxEK1122.A_0017_EPP3744_0041_0016.AI_Inputs_Channel_1.Status/TxPDO_Toggle <-> AI Inputs Channel 1/Status/TxPDO Toggle
//     PlcTask Inputs/GVL_iXlinker.EtherCAT_Master_EPPxxxx.Beckhoff_EPP3xxx.Beckhoff_EPP3xxxEK1122.A_0017_EPP3744_0041_0016.AI_Inputs_Channel_2.Status/TxPDO_Toggle <-> AI Inputs Channel 2/Status/TxPDO Toggle
//     PlcTask Inputs/GVL_iXlinker.EtherCAT_Master_EPPxxxx.Beckhoff_EPP3xxx.Beckhoff_EPP3xxxEK1122.A_0017_EPP3744_0041_0016.AI_Inputs_Channel_3.Status/TxPDO_Toggle <-> AI Inputs Channel 3/Status/TxPDO Toggle
//     PlcTask Inputs/GVL_iXlinker.EtherCAT_Master_EPPxxxx.Beckhoff_EPP3xxx.Beckhoff_EPP3xxxEK1122.A_0017_EPP3744_0041_0016.AI_Inputs_Channel_4.Status/TxPDO_Toggle <-> AI Inputs Channel 4/Status/TxPDO Toggle
//     PlcTask Inputs/GVL_iXlinker.EtherCAT_Master_EPPxxxx.Beckhoff_EPP3xxx.Beckhoff_EPP3xxxEK1122.A_0017_EPP3744_0041_0016.AI_Inputs_Channel_1.Value <-> AI Inputs Channel 1/Value
//     PlcTask Inputs/GVL_iXlinker.EtherCAT_Master_EPPxxxx.Beckhoff_EPP3xxx.Beckhoff_EPP3xxxEK1122.A_0017_EPP3744_0041_0016.AI_Inputs_Channel_2.Value <-> AI Inputs Channel 2/Value
//     PlcTask Inputs/GVL_iXlinker.EtherCAT_Master_EPPxxxx.Beckhoff_EPP3xxx.Beckhoff_EPP3xxxEK1122.A_0017_EPP3744_0041_0016.AI_Inputs_Channel_3.Value <-> AI Inputs Channel 3/Value
//     PlcTask Inputs/GVL_iXlinker.EtherCAT_Master_EPPxxxx.Beckhoff_EPP3xxx.Beckhoff_EPP3xxxEK1122.A_0017_EPP3744_0041_0016.AI_Inputs_Channel_4.Value <-> AI Inputs Channel 4/Value
//     PlcTask Inputs/GVL_iXlinker.EtherCAT_Master_EPPxxxx.Beckhoff_EPP3xxx.Beckhoff_EPP3xxxEK1122.A_0017_EPP3744_0041_0016.DEV_Inputs_Device.Safe_State_Active <-> DEV Inputs Device/Safe State Active
//     PlcTask Inputs/GVL_iXlinker.EtherCAT_Master_EPPxxxx.Beckhoff_EPP3xxx.Beckhoff_EPP3xxxEK1122.A_0017_EPP3744_0041_0016.DEV_Inputs_Device.Sync_error <-> DEV Inputs Device/Sync error
//     PlcTask Inputs/GVL_iXlinker.EtherCAT_Master_EPPxxxx.Beckhoff_EPP3xxx.Beckhoff_EPP3xxxEK1122.A_0017_EPP3744_0041_0016.DEV_Inputs_Device.Undervoltage_Us <-> DEV Inputs Device/Undervoltage Us
//     PlcTask Inputs/GVL_iXlinker.EtherCAT_Master_EPPxxxx.Beckhoff_EPP3xxx.Beckhoff_EPP3xxxEK1122.A_0017_EPP3744_0041_0016.DEV_Inputs_Device.Undervoltage_Up <-> DEV Inputs Device/Undervoltage Up
//     PlcTask Inputs/GVL_iXlinker.EtherCAT_Master_EPPxxxx.Beckhoff_EPP3xxx.Beckhoff_EPP3xxxEK1122.A_0017_EPP3744_0041_0016.DEV_Inputs_Device.TxPDO_Toggle <-> DEV Inputs Device/TxPDO Toggle
//     PlcTask Outputs/GVL_iXlinker.EtherCAT_Master_EPPxxxx.Beckhoff_EPP3xxx.Beckhoff_EPP3xxxEK1122.A_0017_EPP3744_0041_0016.DIG_Outputs.Output[0] <-> DIG Outputs/Output 1
//     PlcTask Outputs/GVL_iXlinker.EtherCAT_Master_EPPxxxx.Beckhoff_EPP3xxx.Beckhoff_EPP3xxxEK1122.A_0017_EPP3744_0041_0016.DIG_Outputs.Output[1] <-> DIG Outputs/Output 2
//     PlcTask Outputs/GVL_iXlinker.EtherCAT_Master_EPPxxxx.Beckhoff_EPP3xxx.Beckhoff_EPP3xxxEK1122.A_0017_EPP3744_0041_0016.DEV_Outputs_Device.Set_safe_state <-> DEV Outputs Device/Set safe state
//     PlcTask Inputs/GVL_iXlinker.EtherCAT_Master_EPPxxxx.Beckhoff_EPP3xxx.Beckhoff_EPP3xxxEK1122.A_0017_EPP3744_0041_0016.WcState.WcState <-> WcState/WcState
//     PlcTask Inputs/GVL_iXlinker.EtherCAT_Master_EPPxxxx.Beckhoff_EPP3xxx.Beckhoff_EPP3xxxEK1122.A_0017_EPP3744_0041_0016.WcState.InputToggle <-> WcState/InputToggle
//     PlcTask Inputs/GVL_iXlinker.EtherCAT_Master_EPPxxxx.Beckhoff_EPP3xxx.Beckhoff_EPP3xxxEK1122.A_0017_EPP3744_0041_0016.InfoData.AdsAddr <-> InfoData/AdsAddr
//     PlcTask Inputs/GVL_iXlinker.EtherCAT_Master_EPPxxxx.Beckhoff_EPP3xxx.Beckhoff_EPP3xxxEK1122.A_0017_EPP3744_0041_0016.InfoData.State <-> InfoData/State
//   PLC/PLC Instance <-> EtherCAT Master EPPxxxx/Beckhoff EPP3xxx/Beckhoff EPP3xxxEK1122/A_0018(EPP3744-0041-0017)
//     PlcTask Inputs/GVL_iXlinker.EtherCAT_Master_EPPxxxx.Beckhoff_EPP3xxx.Beckhoff_EPP3xxxEK1122.A_0018_EPP3744_0041_0017.DIG_Inputs.Input[0] <-> DIG Inputs/Input 1
//     PlcTask Inputs/GVL_iXlinker.EtherCAT_Master_EPPxxxx.Beckhoff_EPP3xxx.Beckhoff_EPP3xxxEK1122.A_0018_EPP3744_0041_0017.DIG_Inputs.Input[1] <-> DIG Inputs/Input 2
//     PlcTask Inputs/GVL_iXlinker.EtherCAT_Master_EPPxxxx.Beckhoff_EPP3xxx.Beckhoff_EPP3xxxEK1122.A_0018_EPP3744_0041_0017.DIG_Inputs.Input[2] <-> DIG Inputs/Input 3
//     PlcTask Inputs/GVL_iXlinker.EtherCAT_Master_EPPxxxx.Beckhoff_EPP3xxx.Beckhoff_EPP3xxxEK1122.A_0018_EPP3744_0041_0017.DIG_Inputs.Input[3] <-> DIG Inputs/Input 4
//     PlcTask Inputs/GVL_iXlinker.EtherCAT_Master_EPPxxxx.Beckhoff_EPP3xxx.Beckhoff_EPP3xxxEK1122.A_0018_EPP3744_0041_0017.DIG_Inputs.Input[4] <-> DIG Inputs/Input 5
//     PlcTask Inputs/GVL_iXlinker.EtherCAT_Master_EPPxxxx.Beckhoff_EPP3xxx.Beckhoff_EPP3xxxEK1122.A_0018_EPP3744_0041_0017.DIG_Inputs.Input[5] <-> DIG Inputs/Input 6
//     PlcTask Inputs/GVL_iXlinker.EtherCAT_Master_EPPxxxx.Beckhoff_EPP3xxx.Beckhoff_EPP3xxxEK1122.A_0018_EPP3744_0041_0017.AI_Inputs_Channel_1.Status/Underrange <-> AI Inputs Channel 1/Status/Underrange
//     PlcTask Inputs/GVL_iXlinker.EtherCAT_Master_EPPxxxx.Beckhoff_EPP3xxx.Beckhoff_EPP3xxxEK1122.A_0018_EPP3744_0041_0017.AI_Inputs_Channel_2.Status/Underrange <-> AI Inputs Channel 2/Status/Underrange
//     PlcTask Inputs/GVL_iXlinker.EtherCAT_Master_EPPxxxx.Beckhoff_EPP3xxx.Beckhoff_EPP3xxxEK1122.A_0018_EPP3744_0041_0017.AI_Inputs_Channel_3.Status/Underrange <-> AI Inputs Channel 3/Status/Underrange
//     PlcTask Inputs/GVL_iXlinker.EtherCAT_Master_EPPxxxx.Beckhoff_EPP3xxx.Beckhoff_EPP3xxxEK1122.A_0018_EPP3744_0041_0017.AI_Inputs_Channel_4.Status/Underrange <-> AI Inputs Channel 4/Status/Underrange
//     PlcTask Inputs/GVL_iXlinker.EtherCAT_Master_EPPxxxx.Beckhoff_EPP3xxx.Beckhoff_EPP3xxxEK1122.A_0018_EPP3744_0041_0017.AI_Inputs_Channel_1.Status/Overrange <-> AI Inputs Channel 1/Status/Overrange
//     PlcTask Inputs/GVL_iXlinker.EtherCAT_Master_EPPxxxx.Beckhoff_EPP3xxx.Beckhoff_EPP3xxxEK1122.A_0018_EPP3744_0041_0017.AI_Inputs_Channel_2.Status/Overrange <-> AI Inputs Channel 2/Status/Overrange
//     PlcTask Inputs/GVL_iXlinker.EtherCAT_Master_EPPxxxx.Beckhoff_EPP3xxx.Beckhoff_EPP3xxxEK1122.A_0018_EPP3744_0041_0017.AI_Inputs_Channel_3.Status/Overrange <-> AI Inputs Channel 3/Status/Overrange
//     PlcTask Inputs/GVL_iXlinker.EtherCAT_Master_EPPxxxx.Beckhoff_EPP3xxx.Beckhoff_EPP3xxxEK1122.A_0018_EPP3744_0041_0017.AI_Inputs_Channel_4.Status/Overrange <-> AI Inputs Channel 4/Status/Overrange
//     PlcTask Inputs/GVL_iXlinker.EtherCAT_Master_EPPxxxx.Beckhoff_EPP3xxx.Beckhoff_EPP3xxxEK1122.A_0018_EPP3744_0041_0017.AI_Inputs_Channel_1.Status/Limit_1 <-> AI Inputs Channel 1/Status/Limit 1
//     PlcTask Inputs/GVL_iXlinker.EtherCAT_Master_EPPxxxx.Beckhoff_EPP3xxx.Beckhoff_EPP3xxxEK1122.A_0018_EPP3744_0041_0017.AI_Inputs_Channel_1.Status/Limit_2 <-> AI Inputs Channel 1/Status/Limit 2
//     PlcTask Inputs/GVL_iXlinker.EtherCAT_Master_EPPxxxx.Beckhoff_EPP3xxx.Beckhoff_EPP3xxxEK1122.A_0018_EPP3744_0041_0017.AI_Inputs_Channel_2.Status/Limit_1 <-> AI Inputs Channel 2/Status/Limit 1
//     PlcTask Inputs/GVL_iXlinker.EtherCAT_Master_EPPxxxx.Beckhoff_EPP3xxx.Beckhoff_EPP3xxxEK1122.A_0018_EPP3744_0041_0017.AI_Inputs_Channel_2.Status/Limit_2 <-> AI Inputs Channel 2/Status/Limit 2
//     PlcTask Inputs/GVL_iXlinker.EtherCAT_Master_EPPxxxx.Beckhoff_EPP3xxx.Beckhoff_EPP3xxxEK1122.A_0018_EPP3744_0041_0017.AI_Inputs_Channel_3.Status/Limit_1 <-> AI Inputs Channel 3/Status/Limit 1
//     PlcTask Inputs/GVL_iXlinker.EtherCAT_Master_EPPxxxx.Beckhoff_EPP3xxx.Beckhoff_EPP3xxxEK1122.A_0018_EPP3744_0041_0017.AI_Inputs_Channel_3.Status/Limit_2 <-> AI Inputs Channel 3/Status/Limit 2
//     PlcTask Inputs/GVL_iXlinker.EtherCAT_Master_EPPxxxx.Beckhoff_EPP3xxx.Beckhoff_EPP3xxxEK1122.A_0018_EPP3744_0041_0017.AI_Inputs_Channel_4.Status/Limit_1 <-> AI Inputs Channel 4/Status/Limit 1
//     PlcTask Inputs/GVL_iXlinker.EtherCAT_Master_EPPxxxx.Beckhoff_EPP3xxx.Beckhoff_EPP3xxxEK1122.A_0018_EPP3744_0041_0017.AI_Inputs_Channel_4.Status/Limit_2 <-> AI Inputs Channel 4/Status/Limit 2
//     PlcTask Inputs/GVL_iXlinker.EtherCAT_Master_EPPxxxx.Beckhoff_EPP3xxx.Beckhoff_EPP3xxxEK1122.A_0018_EPP3744_0041_0017.AI_Inputs_Channel_1.Status/Error <-> AI Inputs Channel 1/Status/Error
//     PlcTask Inputs/GVL_iXlinker.EtherCAT_Master_EPPxxxx.Beckhoff_EPP3xxx.Beckhoff_EPP3xxxEK1122.A_0018_EPP3744_0041_0017.AI_Inputs_Channel_2.Status/Error <-> AI Inputs Channel 2/Status/Error
//     PlcTask Inputs/GVL_iXlinker.EtherCAT_Master_EPPxxxx.Beckhoff_EPP3xxx.Beckhoff_EPP3xxxEK1122.A_0018_EPP3744_0041_0017.AI_Inputs_Channel_3.Status/Error <-> AI Inputs Channel 3/Status/Error
//     PlcTask Inputs/GVL_iXlinker.EtherCAT_Master_EPPxxxx.Beckhoff_EPP3xxx.Beckhoff_EPP3xxxEK1122.A_0018_EPP3744_0041_0017.AI_Inputs_Channel_4.Status/Error <-> AI Inputs Channel 4/Status/Error
//     PlcTask Inputs/GVL_iXlinker.EtherCAT_Master_EPPxxxx.Beckhoff_EPP3xxx.Beckhoff_EPP3xxxEK1122.A_0018_EPP3744_0041_0017.AI_Inputs_Channel_1.Status/TxPDO_State <-> AI Inputs Channel 1/Status/TxPDO State
//     PlcTask Inputs/GVL_iXlinker.EtherCAT_Master_EPPxxxx.Beckhoff_EPP3xxx.Beckhoff_EPP3xxxEK1122.A_0018_EPP3744_0041_0017.AI_Inputs_Channel_2.Status/TxPDO_State <-> AI Inputs Channel 2/Status/TxPDO State
//     PlcTask Inputs/GVL_iXlinker.EtherCAT_Master_EPPxxxx.Beckhoff_EPP3xxx.Beckhoff_EPP3xxxEK1122.A_0018_EPP3744_0041_0017.AI_Inputs_Channel_3.Status/TxPDO_State <-> AI Inputs Channel 3/Status/TxPDO State
//     PlcTask Inputs/GVL_iXlinker.EtherCAT_Master_EPPxxxx.Beckhoff_EPP3xxx.Beckhoff_EPP3xxxEK1122.A_0018_EPP3744_0041_0017.AI_Inputs_Channel_4.Status/TxPDO_State <-> AI Inputs Channel 4/Status/TxPDO State
//     PlcTask Inputs/GVL_iXlinker.EtherCAT_Master_EPPxxxx.Beckhoff_EPP3xxx.Beckhoff_EPP3xxxEK1122.A_0018_EPP3744_0041_0017.AI_Inputs_Channel_1.Status/TxPDO_Toggle <-> AI Inputs Channel 1/Status/TxPDO Toggle
//     PlcTask Inputs/GVL_iXlinker.EtherCAT_Master_EPPxxxx.Beckhoff_EPP3xxx.Beckhoff_EPP3xxxEK1122.A_0018_EPP3744_0041_0017.AI_Inputs_Channel_2.Status/TxPDO_Toggle <-> AI Inputs Channel 2/Status/TxPDO Toggle
//     PlcTask Inputs/GVL_iXlinker.EtherCAT_Master_EPPxxxx.Beckhoff_EPP3xxx.Beckhoff_EPP3xxxEK1122.A_0018_EPP3744_0041_0017.AI_Inputs_Channel_3.Status/TxPDO_Toggle <-> AI Inputs Channel 3/Status/TxPDO Toggle
//     PlcTask Inputs/GVL_iXlinker.EtherCAT_Master_EPPxxxx.Beckhoff_EPP3xxx.Beckhoff_EPP3xxxEK1122.A_0018_EPP3744_0041_0017.AI_Inputs_Channel_4.Status/TxPDO_Toggle <-> AI Inputs Channel 4/Status/TxPDO Toggle
//     PlcTask Inputs/GVL_iXlinker.EtherCAT_Master_EPPxxxx.Beckhoff_EPP3xxx.Beckhoff_EPP3xxxEK1122.A_0018_EPP3744_0041_0017.AI_Inputs_Channel_1.Value <-> AI Inputs Channel 1/Value
//     PlcTask Inputs/GVL_iXlinker.EtherCAT_Master_EPPxxxx.Beckhoff_EPP3xxx.Beckhoff_EPP3xxxEK1122.A_0018_EPP3744_0041_0017.AI_Inputs_Channel_2.Value <-> AI Inputs Channel 2/Value
//     PlcTask Inputs/GVL_iXlinker.EtherCAT_Master_EPPxxxx.Beckhoff_EPP3xxx.Beckhoff_EPP3xxxEK1122.A_0018_EPP3744_0041_0017.AI_Inputs_Channel_3.Value <-> AI Inputs Channel 3/Value
//     PlcTask Inputs/GVL_iXlinker.EtherCAT_Master_EPPxxxx.Beckhoff_EPP3xxx.Beckhoff_EPP3xxxEK1122.A_0018_EPP3744_0041_0017.AI_Inputs_Channel_4.Value <-> AI Inputs Channel 4/Value
//     PlcTask Inputs/GVL_iXlinker.EtherCAT_Master_EPPxxxx.Beckhoff_EPP3xxx.Beckhoff_EPP3xxxEK1122.A_0018_EPP3744_0041_0017.DEV_Inputs_Device.Safe_State_Active <-> DEV Inputs Device/Safe State Active
//     PlcTask Inputs/GVL_iXlinker.EtherCAT_Master_EPPxxxx.Beckhoff_EPP3xxx.Beckhoff_EPP3xxxEK1122.A_0018_EPP3744_0041_0017.DEV_Inputs_Device.Sync_error <-> DEV Inputs Device/Sync error
//     PlcTask Inputs/GVL_iXlinker.EtherCAT_Master_EPPxxxx.Beckhoff_EPP3xxx.Beckhoff_EPP3xxxEK1122.A_0018_EPP3744_0041_0017.DEV_Inputs_Device.Undervoltage_Us <-> DEV Inputs Device/Undervoltage Us
//     PlcTask Inputs/GVL_iXlinker.EtherCAT_Master_EPPxxxx.Beckhoff_EPP3xxx.Beckhoff_EPP3xxxEK1122.A_0018_EPP3744_0041_0017.DEV_Inputs_Device.Undervoltage_Up <-> DEV Inputs Device/Undervoltage Up
//     PlcTask Inputs/GVL_iXlinker.EtherCAT_Master_EPPxxxx.Beckhoff_EPP3xxx.Beckhoff_EPP3xxxEK1122.A_0018_EPP3744_0041_0017.DEV_Inputs_Device.TxPDO_Toggle <-> DEV Inputs Device/TxPDO Toggle
//     PlcTask Outputs/GVL_iXlinker.EtherCAT_Master_EPPxxxx.Beckhoff_EPP3xxx.Beckhoff_EPP3xxxEK1122.A_0018_EPP3744_0041_0017.DIG_Outputs.Output[0] <-> DIG Outputs/Output 1
//     PlcTask Outputs/GVL_iXlinker.EtherCAT_Master_EPPxxxx.Beckhoff_EPP3xxx.Beckhoff_EPP3xxxEK1122.A_0018_EPP3744_0041_0017.DIG_Outputs.Output[1] <-> DIG Outputs/Output 2
//     PlcTask Outputs/GVL_iXlinker.EtherCAT_Master_EPPxxxx.Beckhoff_EPP3xxx.Beckhoff_EPP3xxxEK1122.A_0018_EPP3744_0041_0017.DEV_Outputs_Device.Set_safe_state <-> DEV Outputs Device/Set safe state
//     PlcTask Inputs/GVL_iXlinker.EtherCAT_Master_EPPxxxx.Beckhoff_EPP3xxx.Beckhoff_EPP3xxxEK1122.A_0018_EPP3744_0041_0017.WcState.WcState <-> WcState/WcState
//     PlcTask Inputs/GVL_iXlinker.EtherCAT_Master_EPPxxxx.Beckhoff_EPP3xxx.Beckhoff_EPP3xxxEK1122.A_0018_EPP3744_0041_0017.WcState.InputToggle <-> WcState/InputToggle
//     PlcTask Inputs/GVL_iXlinker.EtherCAT_Master_EPPxxxx.Beckhoff_EPP3xxx.Beckhoff_EPP3xxxEK1122.A_0018_EPP3744_0041_0017.InfoData.AdsAddr <-> InfoData/AdsAddr
//     PlcTask Inputs/GVL_iXlinker.EtherCAT_Master_EPPxxxx.Beckhoff_EPP3xxx.Beckhoff_EPP3xxxEK1122.A_0018_EPP3744_0041_0017.InfoData.State <-> InfoData/State
//   PLC/PLC Instance <-> EtherCAT Master EPPxxxx/Beckhoff EPP3xxx/Beckhoff EPP3xxxEK1122/A_0019(EPP3744-0041-0018)
//     PlcTask Inputs/GVL_iXlinker.EtherCAT_Master_EPPxxxx.Beckhoff_EPP3xxx.Beckhoff_EPP3xxxEK1122.A_0019_EPP3744_0041_0018.DIG_Inputs.Input[0] <-> DIG Inputs/Input 1
//     PlcTask Inputs/GVL_iXlinker.EtherCAT_Master_EPPxxxx.Beckhoff_EPP3xxx.Beckhoff_EPP3xxxEK1122.A_0019_EPP3744_0041_0018.DIG_Inputs.Input[1] <-> DIG Inputs/Input 2
//     PlcTask Inputs/GVL_iXlinker.EtherCAT_Master_EPPxxxx.Beckhoff_EPP3xxx.Beckhoff_EPP3xxxEK1122.A_0019_EPP3744_0041_0018.DIG_Inputs.Input[2] <-> DIG Inputs/Input 3
//     PlcTask Inputs/GVL_iXlinker.EtherCAT_Master_EPPxxxx.Beckhoff_EPP3xxx.Beckhoff_EPP3xxxEK1122.A_0019_EPP3744_0041_0018.DIG_Inputs.Input[3] <-> DIG Inputs/Input 4
//     PlcTask Inputs/GVL_iXlinker.EtherCAT_Master_EPPxxxx.Beckhoff_EPP3xxx.Beckhoff_EPP3xxxEK1122.A_0019_EPP3744_0041_0018.DIG_Inputs.Input[4] <-> DIG Inputs/Input 5
//     PlcTask Inputs/GVL_iXlinker.EtherCAT_Master_EPPxxxx.Beckhoff_EPP3xxx.Beckhoff_EPP3xxxEK1122.A_0019_EPP3744_0041_0018.DIG_Inputs.Input[5] <-> DIG Inputs/Input 6
//     PlcTask Inputs/GVL_iXlinker.EtherCAT_Master_EPPxxxx.Beckhoff_EPP3xxx.Beckhoff_EPP3xxxEK1122.A_0019_EPP3744_0041_0018.AI_Inputs_Channel_1.Status/Underrange <-> AI Inputs Channel 1/Status/Underrange
//     PlcTask Inputs/GVL_iXlinker.EtherCAT_Master_EPPxxxx.Beckhoff_EPP3xxx.Beckhoff_EPP3xxxEK1122.A_0019_EPP3744_0041_0018.AI_Inputs_Channel_2.Status/Underrange <-> AI Inputs Channel 2/Status/Underrange
//     PlcTask Inputs/GVL_iXlinker.EtherCAT_Master_EPPxxxx.Beckhoff_EPP3xxx.Beckhoff_EPP3xxxEK1122.A_0019_EPP3744_0041_0018.AI_Inputs_Channel_3.Status/Underrange <-> AI Inputs Channel 3/Status/Underrange
//     PlcTask Inputs/GVL_iXlinker.EtherCAT_Master_EPPxxxx.Beckhoff_EPP3xxx.Beckhoff_EPP3xxxEK1122.A_0019_EPP3744_0041_0018.AI_Inputs_Channel_4.Status/Underrange <-> AI Inputs Channel 4/Status/Underrange
//     PlcTask Inputs/GVL_iXlinker.EtherCAT_Master_EPPxxxx.Beckhoff_EPP3xxx.Beckhoff_EPP3xxxEK1122.A_0019_EPP3744_0041_0018.AI_Inputs_Channel_1.Status/Overrange <-> AI Inputs Channel 1/Status/Overrange
//     PlcTask Inputs/GVL_iXlinker.EtherCAT_Master_EPPxxxx.Beckhoff_EPP3xxx.Beckhoff_EPP3xxxEK1122.A_0019_EPP3744_0041_0018.AI_Inputs_Channel_2.Status/Overrange <-> AI Inputs Channel 2/Status/Overrange
//     PlcTask Inputs/GVL_iXlinker.EtherCAT_Master_EPPxxxx.Beckhoff_EPP3xxx.Beckhoff_EPP3xxxEK1122.A_0019_EPP3744_0041_0018.AI_Inputs_Channel_3.Status/Overrange <-> AI Inputs Channel 3/Status/Overrange
//     PlcTask Inputs/GVL_iXlinker.EtherCAT_Master_EPPxxxx.Beckhoff_EPP3xxx.Beckhoff_EPP3xxxEK1122.A_0019_EPP3744_0041_0018.AI_Inputs_Channel_4.Status/Overrange <-> AI Inputs Channel 4/Status/Overrange
//     PlcTask Inputs/GVL_iXlinker.EtherCAT_Master_EPPxxxx.Beckhoff_EPP3xxx.Beckhoff_EPP3xxxEK1122.A_0019_EPP3744_0041_0018.AI_Inputs_Channel_1.Status/Limit_1 <-> AI Inputs Channel 1/Status/Limit 1
//     PlcTask Inputs/GVL_iXlinker.EtherCAT_Master_EPPxxxx.Beckhoff_EPP3xxx.Beckhoff_EPP3xxxEK1122.A_0019_EPP3744_0041_0018.AI_Inputs_Channel_1.Status/Limit_2 <-> AI Inputs Channel 1/Status/Limit 2
//     PlcTask Inputs/GVL_iXlinker.EtherCAT_Master_EPPxxxx.Beckhoff_EPP3xxx.Beckhoff_EPP3xxxEK1122.A_0019_EPP3744_0041_0018.AI_Inputs_Channel_2.Status/Limit_1 <-> AI Inputs Channel 2/Status/Limit 1
//     PlcTask Inputs/GVL_iXlinker.EtherCAT_Master_EPPxxxx.Beckhoff_EPP3xxx.Beckhoff_EPP3xxxEK1122.A_0019_EPP3744_0041_0018.AI_Inputs_Channel_2.Status/Limit_2 <-> AI Inputs Channel 2/Status/Limit 2
//     PlcTask Inputs/GVL_iXlinker.EtherCAT_Master_EPPxxxx.Beckhoff_EPP3xxx.Beckhoff_EPP3xxxEK1122.A_0019_EPP3744_0041_0018.AI_Inputs_Channel_3.Status/Limit_1 <-> AI Inputs Channel 3/Status/Limit 1
//     PlcTask Inputs/GVL_iXlinker.EtherCAT_Master_EPPxxxx.Beckhoff_EPP3xxx.Beckhoff_EPP3xxxEK1122.A_0019_EPP3744_0041_0018.AI_Inputs_Channel_3.Status/Limit_2 <-> AI Inputs Channel 3/Status/Limit 2
//     PlcTask Inputs/GVL_iXlinker.EtherCAT_Master_EPPxxxx.Beckhoff_EPP3xxx.Beckhoff_EPP3xxxEK1122.A_0019_EPP3744_0041_0018.AI_Inputs_Channel_4.Status/Limit_1 <-> AI Inputs Channel 4/Status/Limit 1
//     PlcTask Inputs/GVL_iXlinker.EtherCAT_Master_EPPxxxx.Beckhoff_EPP3xxx.Beckhoff_EPP3xxxEK1122.A_0019_EPP3744_0041_0018.AI_Inputs_Channel_4.Status/Limit_2 <-> AI Inputs Channel 4/Status/Limit 2
//     PlcTask Inputs/GVL_iXlinker.EtherCAT_Master_EPPxxxx.Beckhoff_EPP3xxx.Beckhoff_EPP3xxxEK1122.A_0019_EPP3744_0041_0018.AI_Inputs_Channel_1.Status/Error <-> AI Inputs Channel 1/Status/Error
//     PlcTask Inputs/GVL_iXlinker.EtherCAT_Master_EPPxxxx.Beckhoff_EPP3xxx.Beckhoff_EPP3xxxEK1122.A_0019_EPP3744_0041_0018.AI_Inputs_Channel_2.Status/Error <-> AI Inputs Channel 2/Status/Error
//     PlcTask Inputs/GVL_iXlinker.EtherCAT_Master_EPPxxxx.Beckhoff_EPP3xxx.Beckhoff_EPP3xxxEK1122.A_0019_EPP3744_0041_0018.AI_Inputs_Channel_3.Status/Error <-> AI Inputs Channel 3/Status/Error
//     PlcTask Inputs/GVL_iXlinker.EtherCAT_Master_EPPxxxx.Beckhoff_EPP3xxx.Beckhoff_EPP3xxxEK1122.A_0019_EPP3744_0041_0018.AI_Inputs_Channel_4.Status/Error <-> AI Inputs Channel 4/Status/Error
//     PlcTask Inputs/GVL_iXlinker.EtherCAT_Master_EPPxxxx.Beckhoff_EPP3xxx.Beckhoff_EPP3xxxEK1122.A_0019_EPP3744_0041_0018.AI_Inputs_Channel_1.Status/TxPDO_State <-> AI Inputs Channel 1/Status/TxPDO State
//     PlcTask Inputs/GVL_iXlinker.EtherCAT_Master_EPPxxxx.Beckhoff_EPP3xxx.Beckhoff_EPP3xxxEK1122.A_0019_EPP3744_0041_0018.AI_Inputs_Channel_2.Status/TxPDO_State <-> AI Inputs Channel 2/Status/TxPDO State
//     PlcTask Inputs/GVL_iXlinker.EtherCAT_Master_EPPxxxx.Beckhoff_EPP3xxx.Beckhoff_EPP3xxxEK1122.A_0019_EPP3744_0041_0018.AI_Inputs_Channel_3.Status/TxPDO_State <-> AI Inputs Channel 3/Status/TxPDO State
//     PlcTask Inputs/GVL_iXlinker.EtherCAT_Master_EPPxxxx.Beckhoff_EPP3xxx.Beckhoff_EPP3xxxEK1122.A_0019_EPP3744_0041_0018.AI_Inputs_Channel_4.Status/TxPDO_State <-> AI Inputs Channel 4/Status/TxPDO State
//     PlcTask Inputs/GVL_iXlinker.EtherCAT_Master_EPPxxxx.Beckhoff_EPP3xxx.Beckhoff_EPP3xxxEK1122.A_0019_EPP3744_0041_0018.AI_Inputs_Channel_1.Status/TxPDO_Toggle <-> AI Inputs Channel 1/Status/TxPDO Toggle
//     PlcTask Inputs/GVL_iXlinker.EtherCAT_Master_EPPxxxx.Beckhoff_EPP3xxx.Beckhoff_EPP3xxxEK1122.A_0019_EPP3744_0041_0018.AI_Inputs_Channel_2.Status/TxPDO_Toggle <-> AI Inputs Channel 2/Status/TxPDO Toggle
//     PlcTask Inputs/GVL_iXlinker.EtherCAT_Master_EPPxxxx.Beckhoff_EPP3xxx.Beckhoff_EPP3xxxEK1122.A_0019_EPP3744_0041_0018.AI_Inputs_Channel_3.Status/TxPDO_Toggle <-> AI Inputs Channel 3/Status/TxPDO Toggle
//     PlcTask Inputs/GVL_iXlinker.EtherCAT_Master_EPPxxxx.Beckhoff_EPP3xxx.Beckhoff_EPP3xxxEK1122.A_0019_EPP3744_0041_0018.AI_Inputs_Channel_4.Status/TxPDO_Toggle <-> AI Inputs Channel 4/Status/TxPDO Toggle
//     PlcTask Inputs/GVL_iXlinker.EtherCAT_Master_EPPxxxx.Beckhoff_EPP3xxx.Beckhoff_EPP3xxxEK1122.A_0019_EPP3744_0041_0018.AI_Inputs_Channel_1.Value <-> AI Inputs Channel 1/Value
//     PlcTask Inputs/GVL_iXlinker.EtherCAT_Master_EPPxxxx.Beckhoff_EPP3xxx.Beckhoff_EPP3xxxEK1122.A_0019_EPP3744_0041_0018.AI_Inputs_Channel_2.Value <-> AI Inputs Channel 2/Value
//     PlcTask Inputs/GVL_iXlinker.EtherCAT_Master_EPPxxxx.Beckhoff_EPP3xxx.Beckhoff_EPP3xxxEK1122.A_0019_EPP3744_0041_0018.AI_Inputs_Channel_3.Value <-> AI Inputs Channel 3/Value
//     PlcTask Inputs/GVL_iXlinker.EtherCAT_Master_EPPxxxx.Beckhoff_EPP3xxx.Beckhoff_EPP3xxxEK1122.A_0019_EPP3744_0041_0018.AI_Inputs_Channel_4.Value <-> AI Inputs Channel 4/Value
//     PlcTask Inputs/GVL_iXlinker.EtherCAT_Master_EPPxxxx.Beckhoff_EPP3xxx.Beckhoff_EPP3xxxEK1122.A_0019_EPP3744_0041_0018.DEV_Inputs_Device.Safe_State_Active <-> DEV Inputs Device/Safe State Active
//     PlcTask Inputs/GVL_iXlinker.EtherCAT_Master_EPPxxxx.Beckhoff_EPP3xxx.Beckhoff_EPP3xxxEK1122.A_0019_EPP3744_0041_0018.DEV_Inputs_Device.Sync_error <-> DEV Inputs Device/Sync error
//     PlcTask Inputs/GVL_iXlinker.EtherCAT_Master_EPPxxxx.Beckhoff_EPP3xxx.Beckhoff_EPP3xxxEK1122.A_0019_EPP3744_0041_0018.DEV_Inputs_Device.Undervoltage_Us <-> DEV Inputs Device/Undervoltage Us
//     PlcTask Inputs/GVL_iXlinker.EtherCAT_Master_EPPxxxx.Beckhoff_EPP3xxx.Beckhoff_EPP3xxxEK1122.A_0019_EPP3744_0041_0018.DEV_Inputs_Device.Undervoltage_Up <-> DEV Inputs Device/Undervoltage Up
//     PlcTask Inputs/GVL_iXlinker.EtherCAT_Master_EPPxxxx.Beckhoff_EPP3xxx.Beckhoff_EPP3xxxEK1122.A_0019_EPP3744_0041_0018.DEV_Inputs_Device.TxPDO_Toggle <-> DEV Inputs Device/TxPDO Toggle
//     PlcTask Outputs/GVL_iXlinker.EtherCAT_Master_EPPxxxx.Beckhoff_EPP3xxx.Beckhoff_EPP3xxxEK1122.A_0019_EPP3744_0041_0018.DIG_Outputs.Output[0] <-> DIG Outputs/Output 1
//     PlcTask Outputs/GVL_iXlinker.EtherCAT_Master_EPPxxxx.Beckhoff_EPP3xxx.Beckhoff_EPP3xxxEK1122.A_0019_EPP3744_0041_0018.DIG_Outputs.Output[1] <-> DIG Outputs/Output 2
//     PlcTask Outputs/GVL_iXlinker.EtherCAT_Master_EPPxxxx.Beckhoff_EPP3xxx.Beckhoff_EPP3xxxEK1122.A_0019_EPP3744_0041_0018.DEV_Outputs_Device.Set_safe_state <-> DEV Outputs Device/Set safe state
//     PlcTask Inputs/GVL_iXlinker.EtherCAT_Master_EPPxxxx.Beckhoff_EPP3xxx.Beckhoff_EPP3xxxEK1122.A_0019_EPP3744_0041_0018.WcState.WcState <-> WcState/WcState
//     PlcTask Inputs/GVL_iXlinker.EtherCAT_Master_EPPxxxx.Beckhoff_EPP3xxx.Beckhoff_EPP3xxxEK1122.A_0019_EPP3744_0041_0018.WcState.InputToggle <-> WcState/InputToggle
//     PlcTask Inputs/GVL_iXlinker.EtherCAT_Master_EPPxxxx.Beckhoff_EPP3xxx.Beckhoff_EPP3xxxEK1122.A_0019_EPP3744_0041_0018.InfoData.AdsAddr <-> InfoData/AdsAddr
//     PlcTask Inputs/GVL_iXlinker.EtherCAT_Master_EPPxxxx.Beckhoff_EPP3xxx.Beckhoff_EPP3xxxEK1122.A_0019_EPP3744_0041_0018.InfoData.State <-> InfoData/State
//   PLC/PLC Instance <-> EtherCAT Master EPPxxxx/Beckhoff EPP3xxx/Beckhoff EPP3xxxEK1122/A_0020(EPP3744-1041-0016)
//     PlcTask Inputs/GVL_iXlinker.EtherCAT_Master_EPPxxxx.Beckhoff_EPP3xxx.Beckhoff_EPP3xxxEK1122.A_0020_EPP3744_1041_0016.DIG_Inputs.Input[0] <-> DIG Inputs/Input 1
//     PlcTask Inputs/GVL_iXlinker.EtherCAT_Master_EPPxxxx.Beckhoff_EPP3xxx.Beckhoff_EPP3xxxEK1122.A_0020_EPP3744_1041_0016.DIG_Inputs.Input[1] <-> DIG Inputs/Input 2
//     PlcTask Inputs/GVL_iXlinker.EtherCAT_Master_EPPxxxx.Beckhoff_EPP3xxx.Beckhoff_EPP3xxxEK1122.A_0020_EPP3744_1041_0016.DIG_Inputs.Input[2] <-> DIG Inputs/Input 3
//     PlcTask Inputs/GVL_iXlinker.EtherCAT_Master_EPPxxxx.Beckhoff_EPP3xxx.Beckhoff_EPP3xxxEK1122.A_0020_EPP3744_1041_0016.DIG_Inputs.Input[3] <-> DIG Inputs/Input 4
//     PlcTask Inputs/GVL_iXlinker.EtherCAT_Master_EPPxxxx.Beckhoff_EPP3xxx.Beckhoff_EPP3xxxEK1122.A_0020_EPP3744_1041_0016.DIG_Inputs.Input[4] <-> DIG Inputs/Input 5
//     PlcTask Inputs/GVL_iXlinker.EtherCAT_Master_EPPxxxx.Beckhoff_EPP3xxx.Beckhoff_EPP3xxxEK1122.A_0020_EPP3744_1041_0016.DIG_Inputs.Input[5] <-> DIG Inputs/Input 6
//     PlcTask Inputs/GVL_iXlinker.EtherCAT_Master_EPPxxxx.Beckhoff_EPP3xxx.Beckhoff_EPP3xxxEK1122.A_0020_EPP3744_1041_0016.AI_Inputs_Channel_1.Status/Underrange <-> AI Inputs Channel 1/Status/Underrange
//     PlcTask Inputs/GVL_iXlinker.EtherCAT_Master_EPPxxxx.Beckhoff_EPP3xxx.Beckhoff_EPP3xxxEK1122.A_0020_EPP3744_1041_0016.AI_Inputs_Channel_2.Status/Underrange <-> AI Inputs Channel 2/Status/Underrange
//     PlcTask Inputs/GVL_iXlinker.EtherCAT_Master_EPPxxxx.Beckhoff_EPP3xxx.Beckhoff_EPP3xxxEK1122.A_0020_EPP3744_1041_0016.AI_Inputs_Channel_3.Status/Underrange <-> AI Inputs Channel 3/Status/Underrange
//     PlcTask Inputs/GVL_iXlinker.EtherCAT_Master_EPPxxxx.Beckhoff_EPP3xxx.Beckhoff_EPP3xxxEK1122.A_0020_EPP3744_1041_0016.AI_Inputs_Channel_4.Status/Underrange <-> AI Inputs Channel 4/Status/Underrange
//     PlcTask Inputs/GVL_iXlinker.EtherCAT_Master_EPPxxxx.Beckhoff_EPP3xxx.Beckhoff_EPP3xxxEK1122.A_0020_EPP3744_1041_0016.AI_Inputs_Channel_1.Status/Overrange <-> AI Inputs Channel 1/Status/Overrange
//     PlcTask Inputs/GVL_iXlinker.EtherCAT_Master_EPPxxxx.Beckhoff_EPP3xxx.Beckhoff_EPP3xxxEK1122.A_0020_EPP3744_1041_0016.AI_Inputs_Channel_2.Status/Overrange <-> AI Inputs Channel 2/Status/Overrange
//     PlcTask Inputs/GVL_iXlinker.EtherCAT_Master_EPPxxxx.Beckhoff_EPP3xxx.Beckhoff_EPP3xxxEK1122.A_0020_EPP3744_1041_0016.AI_Inputs_Channel_3.Status/Overrange <-> AI Inputs Channel 3/Status/Overrange
//     PlcTask Inputs/GVL_iXlinker.EtherCAT_Master_EPPxxxx.Beckhoff_EPP3xxx.Beckhoff_EPP3xxxEK1122.A_0020_EPP3744_1041_0016.AI_Inputs_Channel_4.Status/Overrange <-> AI Inputs Channel 4/Status/Overrange
//     PlcTask Inputs/GVL_iXlinker.EtherCAT_Master_EPPxxxx.Beckhoff_EPP3xxx.Beckhoff_EPP3xxxEK1122.A_0020_EPP3744_1041_0016.AI_Inputs_Channel_1.Status/Limit_1 <-> AI Inputs Channel 1/Status/Limit 1
//     PlcTask Inputs/GVL_iXlinker.EtherCAT_Master_EPPxxxx.Beckhoff_EPP3xxx.Beckhoff_EPP3xxxEK1122.A_0020_EPP3744_1041_0016.AI_Inputs_Channel_1.Status/Limit_2 <-> AI Inputs Channel 1/Status/Limit 2
//     PlcTask Inputs/GVL_iXlinker.EtherCAT_Master_EPPxxxx.Beckhoff_EPP3xxx.Beckhoff_EPP3xxxEK1122.A_0020_EPP3744_1041_0016.AI_Inputs_Channel_2.Status/Limit_1 <-> AI Inputs Channel 2/Status/Limit 1
//     PlcTask Inputs/GVL_iXlinker.EtherCAT_Master_EPPxxxx.Beckhoff_EPP3xxx.Beckhoff_EPP3xxxEK1122.A_0020_EPP3744_1041_0016.AI_Inputs_Channel_2.Status/Limit_2 <-> AI Inputs Channel 2/Status/Limit 2
//     PlcTask Inputs/GVL_iXlinker.EtherCAT_Master_EPPxxxx.Beckhoff_EPP3xxx.Beckhoff_EPP3xxxEK1122.A_0020_EPP3744_1041_0016.AI_Inputs_Channel_3.Status/Limit_1 <-> AI Inputs Channel 3/Status/Limit 1
//     PlcTask Inputs/GVL_iXlinker.EtherCAT_Master_EPPxxxx.Beckhoff_EPP3xxx.Beckhoff_EPP3xxxEK1122.A_0020_EPP3744_1041_0016.AI_Inputs_Channel_3.Status/Limit_2 <-> AI Inputs Channel 3/Status/Limit 2
//     PlcTask Inputs/GVL_iXlinker.EtherCAT_Master_EPPxxxx.Beckhoff_EPP3xxx.Beckhoff_EPP3xxxEK1122.A_0020_EPP3744_1041_0016.AI_Inputs_Channel_4.Status/Limit_1 <-> AI Inputs Channel 4/Status/Limit 1
//     PlcTask Inputs/GVL_iXlinker.EtherCAT_Master_EPPxxxx.Beckhoff_EPP3xxx.Beckhoff_EPP3xxxEK1122.A_0020_EPP3744_1041_0016.AI_Inputs_Channel_4.Status/Limit_2 <-> AI Inputs Channel 4/Status/Limit 2
//     PlcTask Inputs/GVL_iXlinker.EtherCAT_Master_EPPxxxx.Beckhoff_EPP3xxx.Beckhoff_EPP3xxxEK1122.A_0020_EPP3744_1041_0016.AI_Inputs_Channel_1.Status/Error <-> AI Inputs Channel 1/Status/Error
//     PlcTask Inputs/GVL_iXlinker.EtherCAT_Master_EPPxxxx.Beckhoff_EPP3xxx.Beckhoff_EPP3xxxEK1122.A_0020_EPP3744_1041_0016.AI_Inputs_Channel_2.Status/Error <-> AI Inputs Channel 2/Status/Error
//     PlcTask Inputs/GVL_iXlinker.EtherCAT_Master_EPPxxxx.Beckhoff_EPP3xxx.Beckhoff_EPP3xxxEK1122.A_0020_EPP3744_1041_0016.AI_Inputs_Channel_3.Status/Error <-> AI Inputs Channel 3/Status/Error
//     PlcTask Inputs/GVL_iXlinker.EtherCAT_Master_EPPxxxx.Beckhoff_EPP3xxx.Beckhoff_EPP3xxxEK1122.A_0020_EPP3744_1041_0016.AI_Inputs_Channel_4.Status/Error <-> AI Inputs Channel 4/Status/Error
//     PlcTask Inputs/GVL_iXlinker.EtherCAT_Master_EPPxxxx.Beckhoff_EPP3xxx.Beckhoff_EPP3xxxEK1122.A_0020_EPP3744_1041_0016.AI_Inputs_Channel_1.Status/TxPDO_State <-> AI Inputs Channel 1/Status/TxPDO State
//     PlcTask Inputs/GVL_iXlinker.EtherCAT_Master_EPPxxxx.Beckhoff_EPP3xxx.Beckhoff_EPP3xxxEK1122.A_0020_EPP3744_1041_0016.AI_Inputs_Channel_2.Status/TxPDO_State <-> AI Inputs Channel 2/Status/TxPDO State
//     PlcTask Inputs/GVL_iXlinker.EtherCAT_Master_EPPxxxx.Beckhoff_EPP3xxx.Beckhoff_EPP3xxxEK1122.A_0020_EPP3744_1041_0016.AI_Inputs_Channel_3.Status/TxPDO_State <-> AI Inputs Channel 3/Status/TxPDO State
//     PlcTask Inputs/GVL_iXlinker.EtherCAT_Master_EPPxxxx.Beckhoff_EPP3xxx.Beckhoff_EPP3xxxEK1122.A_0020_EPP3744_1041_0016.AI_Inputs_Channel_4.Status/TxPDO_State <-> AI Inputs Channel 4/Status/TxPDO State
//     PlcTask Inputs/GVL_iXlinker.EtherCAT_Master_EPPxxxx.Beckhoff_EPP3xxx.Beckhoff_EPP3xxxEK1122.A_0020_EPP3744_1041_0016.AI_Inputs_Channel_1.Status/TxPDO_Toggle <-> AI Inputs Channel 1/Status/TxPDO Toggle
//     PlcTask Inputs/GVL_iXlinker.EtherCAT_Master_EPPxxxx.Beckhoff_EPP3xxx.Beckhoff_EPP3xxxEK1122.A_0020_EPP3744_1041_0016.AI_Inputs_Channel_2.Status/TxPDO_Toggle <-> AI Inputs Channel 2/Status/TxPDO Toggle
//     PlcTask Inputs/GVL_iXlinker.EtherCAT_Master_EPPxxxx.Beckhoff_EPP3xxx.Beckhoff_EPP3xxxEK1122.A_0020_EPP3744_1041_0016.AI_Inputs_Channel_3.Status/TxPDO_Toggle <-> AI Inputs Channel 3/Status/TxPDO Toggle
//     PlcTask Inputs/GVL_iXlinker.EtherCAT_Master_EPPxxxx.Beckhoff_EPP3xxx.Beckhoff_EPP3xxxEK1122.A_0020_EPP3744_1041_0016.AI_Inputs_Channel_4.Status/TxPDO_Toggle <-> AI Inputs Channel 4/Status/TxPDO Toggle
//     PlcTask Inputs/GVL_iXlinker.EtherCAT_Master_EPPxxxx.Beckhoff_EPP3xxx.Beckhoff_EPP3xxxEK1122.A_0020_EPP3744_1041_0016.AI_Inputs_Channel_1.Value <-> AI Inputs Channel 1/Value
//     PlcTask Inputs/GVL_iXlinker.EtherCAT_Master_EPPxxxx.Beckhoff_EPP3xxx.Beckhoff_EPP3xxxEK1122.A_0020_EPP3744_1041_0016.AI_Inputs_Channel_2.Value <-> AI Inputs Channel 2/Value
//     PlcTask Inputs/GVL_iXlinker.EtherCAT_Master_EPPxxxx.Beckhoff_EPP3xxx.Beckhoff_EPP3xxxEK1122.A_0020_EPP3744_1041_0016.AI_Inputs_Channel_3.Value <-> AI Inputs Channel 3/Value
//     PlcTask Inputs/GVL_iXlinker.EtherCAT_Master_EPPxxxx.Beckhoff_EPP3xxx.Beckhoff_EPP3xxxEK1122.A_0020_EPP3744_1041_0016.AI_Inputs_Channel_4.Value <-> AI Inputs Channel 4/Value
//     PlcTask Inputs/GVL_iXlinker.EtherCAT_Master_EPPxxxx.Beckhoff_EPP3xxx.Beckhoff_EPP3xxxEK1122.A_0020_EPP3744_1041_0016.DEV_Inputs_Device.Safe_State_Active <-> DEV Inputs Device/Safe State Active
//     PlcTask Inputs/GVL_iXlinker.EtherCAT_Master_EPPxxxx.Beckhoff_EPP3xxx.Beckhoff_EPP3xxxEK1122.A_0020_EPP3744_1041_0016.DEV_Inputs_Device.Sync_error <-> DEV Inputs Device/Sync error
//     PlcTask Inputs/GVL_iXlinker.EtherCAT_Master_EPPxxxx.Beckhoff_EPP3xxx.Beckhoff_EPP3xxxEK1122.A_0020_EPP3744_1041_0016.DEV_Inputs_Device.Undervoltage_Us <-> DEV Inputs Device/Undervoltage Us
//     PlcTask Inputs/GVL_iXlinker.EtherCAT_Master_EPPxxxx.Beckhoff_EPP3xxx.Beckhoff_EPP3xxxEK1122.A_0020_EPP3744_1041_0016.DEV_Inputs_Device.Undervoltage_Up <-> DEV Inputs Device/Undervoltage Up
//     PlcTask Inputs/GVL_iXlinker.EtherCAT_Master_EPPxxxx.Beckhoff_EPP3xxx.Beckhoff_EPP3xxxEK1122.A_0020_EPP3744_1041_0016.DEV_Inputs_Device.TxPDO_Toggle <-> DEV Inputs Device/TxPDO Toggle
//     PlcTask Outputs/GVL_iXlinker.EtherCAT_Master_EPPxxxx.Beckhoff_EPP3xxx.Beckhoff_EPP3xxxEK1122.A_0020_EPP3744_1041_0016.DIG_Outputs.Output[0] <-> DIG Outputs/Output 1
//     PlcTask Outputs/GVL_iXlinker.EtherCAT_Master_EPPxxxx.Beckhoff_EPP3xxx.Beckhoff_EPP3xxxEK1122.A_0020_EPP3744_1041_0016.DIG_Outputs.Output[1] <-> DIG Outputs/Output 2
//     PlcTask Outputs/GVL_iXlinker.EtherCAT_Master_EPPxxxx.Beckhoff_EPP3xxx.Beckhoff_EPP3xxxEK1122.A_0020_EPP3744_1041_0016.DEV_Outputs_Device.Set_safe_state <-> DEV Outputs Device/Set safe state
//     PlcTask Inputs/GVL_iXlinker.EtherCAT_Master_EPPxxxx.Beckhoff_EPP3xxx.Beckhoff_EPP3xxxEK1122.A_0020_EPP3744_1041_0016.WcState.WcState <-> WcState/WcState
//     PlcTask Inputs/GVL_iXlinker.EtherCAT_Master_EPPxxxx.Beckhoff_EPP3xxx.Beckhoff_EPP3xxxEK1122.A_0020_EPP3744_1041_0016.WcState.InputToggle <-> WcState/InputToggle
//     PlcTask Inputs/GVL_iXlinker.EtherCAT_Master_EPPxxxx.Beckhoff_EPP3xxx.Beckhoff_EPP3xxxEK1122.A_0020_EPP3744_1041_0016.InfoData.AdsAddr <-> InfoData/AdsAddr
//     PlcTask Inputs/GVL_iXlinker.EtherCAT_Master_EPPxxxx.Beckhoff_EPP3xxx.Beckhoff_EPP3xxxEK1122.A_0020_EPP3744_1041_0016.InfoData.State <-> InfoData/State
//   PLC/PLC Instance <-> EtherCAT Master EPPxxxx/Beckhoff EPP3xxx/Beckhoff EPP3xxxEK1122/A_0021(EPP3744-1041-0017)
//     PlcTask Inputs/GVL_iXlinker.EtherCAT_Master_EPPxxxx.Beckhoff_EPP3xxx.Beckhoff_EPP3xxxEK1122.A_0021_EPP3744_1041_0017.DIG_Inputs.Input[0] <-> DIG Inputs/Input 1
//     PlcTask Inputs/GVL_iXlinker.EtherCAT_Master_EPPxxxx.Beckhoff_EPP3xxx.Beckhoff_EPP3xxxEK1122.A_0021_EPP3744_1041_0017.DIG_Inputs.Input[1] <-> DIG Inputs/Input 2
//     PlcTask Inputs/GVL_iXlinker.EtherCAT_Master_EPPxxxx.Beckhoff_EPP3xxx.Beckhoff_EPP3xxxEK1122.A_0021_EPP3744_1041_0017.DIG_Inputs.Input[2] <-> DIG Inputs/Input 3
//     PlcTask Inputs/GVL_iXlinker.EtherCAT_Master_EPPxxxx.Beckhoff_EPP3xxx.Beckhoff_EPP3xxxEK1122.A_0021_EPP3744_1041_0017.DIG_Inputs.Input[3] <-> DIG Inputs/Input 4
//     PlcTask Inputs/GVL_iXlinker.EtherCAT_Master_EPPxxxx.Beckhoff_EPP3xxx.Beckhoff_EPP3xxxEK1122.A_0021_EPP3744_1041_0017.DIG_Inputs.Input[4] <-> DIG Inputs/Input 5
//     PlcTask Inputs/GVL_iXlinker.EtherCAT_Master_EPPxxxx.Beckhoff_EPP3xxx.Beckhoff_EPP3xxxEK1122.A_0021_EPP3744_1041_0017.DIG_Inputs.Input[5] <-> DIG Inputs/Input 6
//     PlcTask Inputs/GVL_iXlinker.EtherCAT_Master_EPPxxxx.Beckhoff_EPP3xxx.Beckhoff_EPP3xxxEK1122.A_0021_EPP3744_1041_0017.AI_Inputs_Channel_1.Status/Underrange <-> AI Inputs Channel 1/Status/Underrange
//     PlcTask Inputs/GVL_iXlinker.EtherCAT_Master_EPPxxxx.Beckhoff_EPP3xxx.Beckhoff_EPP3xxxEK1122.A_0021_EPP3744_1041_0017.AI_Inputs_Channel_2.Status/Underrange <-> AI Inputs Channel 2/Status/Underrange
//     PlcTask Inputs/GVL_iXlinker.EtherCAT_Master_EPPxxxx.Beckhoff_EPP3xxx.Beckhoff_EPP3xxxEK1122.A_0021_EPP3744_1041_0017.AI_Inputs_Channel_3.Status/Underrange <-> AI Inputs Channel 3/Status/Underrange
//     PlcTask Inputs/GVL_iXlinker.EtherCAT_Master_EPPxxxx.Beckhoff_EPP3xxx.Beckhoff_EPP3xxxEK1122.A_0021_EPP3744_1041_0017.AI_Inputs_Channel_4.Status/Underrange <-> AI Inputs Channel 4/Status/Underrange
//     PlcTask Inputs/GVL_iXlinker.EtherCAT_Master_EPPxxxx.Beckhoff_EPP3xxx.Beckhoff_EPP3xxxEK1122.A_0021_EPP3744_1041_0017.AI_Inputs_Channel_1.Status/Overrange <-> AI Inputs Channel 1/Status/Overrange
//     PlcTask Inputs/GVL_iXlinker.EtherCAT_Master_EPPxxxx.Beckhoff_EPP3xxx.Beckhoff_EPP3xxxEK1122.A_0021_EPP3744_1041_0017.AI_Inputs_Channel_2.Status/Overrange <-> AI Inputs Channel 2/Status/Overrange
//     PlcTask Inputs/GVL_iXlinker.EtherCAT_Master_EPPxxxx.Beckhoff_EPP3xxx.Beckhoff_EPP3xxxEK1122.A_0021_EPP3744_1041_0017.AI_Inputs_Channel_3.Status/Overrange <-> AI Inputs Channel 3/Status/Overrange
//     PlcTask Inputs/GVL_iXlinker.EtherCAT_Master_EPPxxxx.Beckhoff_EPP3xxx.Beckhoff_EPP3xxxEK1122.A_0021_EPP3744_1041_0017.AI_Inputs_Channel_4.Status/Overrange <-> AI Inputs Channel 4/Status/Overrange
//     PlcTask Inputs/GVL_iXlinker.EtherCAT_Master_EPPxxxx.Beckhoff_EPP3xxx.Beckhoff_EPP3xxxEK1122.A_0021_EPP3744_1041_0017.AI_Inputs_Channel_1.Status/Limit_1 <-> AI Inputs Channel 1/Status/Limit 1
//     PlcTask Inputs/GVL_iXlinker.EtherCAT_Master_EPPxxxx.Beckhoff_EPP3xxx.Beckhoff_EPP3xxxEK1122.A_0021_EPP3744_1041_0017.AI_Inputs_Channel_1.Status/Limit_2 <-> AI Inputs Channel 1/Status/Limit 2
//     PlcTask Inputs/GVL_iXlinker.EtherCAT_Master_EPPxxxx.Beckhoff_EPP3xxx.Beckhoff_EPP3xxxEK1122.A_0021_EPP3744_1041_0017.AI_Inputs_Channel_2.Status/Limit_1 <-> AI Inputs Channel 2/Status/Limit 1
//     PlcTask Inputs/GVL_iXlinker.EtherCAT_Master_EPPxxxx.Beckhoff_EPP3xxx.Beckhoff_EPP3xxxEK1122.A_0021_EPP3744_1041_0017.AI_Inputs_Channel_2.Status/Limit_2 <-> AI Inputs Channel 2/Status/Limit 2
//     PlcTask Inputs/GVL_iXlinker.EtherCAT_Master_EPPxxxx.Beckhoff_EPP3xxx.Beckhoff_EPP3xxxEK1122.A_0021_EPP3744_1041_0017.AI_Inputs_Channel_3.Status/Limit_1 <-> AI Inputs Channel 3/Status/Limit 1
//     PlcTask Inputs/GVL_iXlinker.EtherCAT_Master_EPPxxxx.Beckhoff_EPP3xxx.Beckhoff_EPP3xxxEK1122.A_0021_EPP3744_1041_0017.AI_Inputs_Channel_3.Status/Limit_2 <-> AI Inputs Channel 3/Status/Limit 2
//     PlcTask Inputs/GVL_iXlinker.EtherCAT_Master_EPPxxxx.Beckhoff_EPP3xxx.Beckhoff_EPP3xxxEK1122.A_0021_EPP3744_1041_0017.AI_Inputs_Channel_4.Status/Limit_1 <-> AI Inputs Channel 4/Status/Limit 1
//     PlcTask Inputs/GVL_iXlinker.EtherCAT_Master_EPPxxxx.Beckhoff_EPP3xxx.Beckhoff_EPP3xxxEK1122.A_0021_EPP3744_1041_0017.AI_Inputs_Channel_4.Status/Limit_2 <-> AI Inputs Channel 4/Status/Limit 2
//     PlcTask Inputs/GVL_iXlinker.EtherCAT_Master_EPPxxxx.Beckhoff_EPP3xxx.Beckhoff_EPP3xxxEK1122.A_0021_EPP3744_1041_0017.AI_Inputs_Channel_1.Status/Error <-> AI Inputs Channel 1/Status/Error
//     PlcTask Inputs/GVL_iXlinker.EtherCAT_Master_EPPxxxx.Beckhoff_EPP3xxx.Beckhoff_EPP3xxxEK1122.A_0021_EPP3744_1041_0017.AI_Inputs_Channel_2.Status/Error <-> AI Inputs Channel 2/Status/Error
//     PlcTask Inputs/GVL_iXlinker.EtherCAT_Master_EPPxxxx.Beckhoff_EPP3xxx.Beckhoff_EPP3xxxEK1122.A_0021_EPP3744_1041_0017.AI_Inputs_Channel_3.Status/Error <-> AI Inputs Channel 3/Status/Error
//     PlcTask Inputs/GVL_iXlinker.EtherCAT_Master_EPPxxxx.Beckhoff_EPP3xxx.Beckhoff_EPP3xxxEK1122.A_0021_EPP3744_1041_0017.AI_Inputs_Channel_4.Status/Error <-> AI Inputs Channel 4/Status/Error
//     PlcTask Inputs/GVL_iXlinker.EtherCAT_Master_EPPxxxx.Beckhoff_EPP3xxx.Beckhoff_EPP3xxxEK1122.A_0021_EPP3744_1041_0017.AI_Inputs_Channel_1.Status/TxPDO_State <-> AI Inputs Channel 1/Status/TxPDO State
//     PlcTask Inputs/GVL_iXlinker.EtherCAT_Master_EPPxxxx.Beckhoff_EPP3xxx.Beckhoff_EPP3xxxEK1122.A_0021_EPP3744_1041_0017.AI_Inputs_Channel_2.Status/TxPDO_State <-> AI Inputs Channel 2/Status/TxPDO State
//     PlcTask Inputs/GVL_iXlinker.EtherCAT_Master_EPPxxxx.Beckhoff_EPP3xxx.Beckhoff_EPP3xxxEK1122.A_0021_EPP3744_1041_0017.AI_Inputs_Channel_3.Status/TxPDO_State <-> AI Inputs Channel 3/Status/TxPDO State
//     PlcTask Inputs/GVL_iXlinker.EtherCAT_Master_EPPxxxx.Beckhoff_EPP3xxx.Beckhoff_EPP3xxxEK1122.A_0021_EPP3744_1041_0017.AI_Inputs_Channel_4.Status/TxPDO_State <-> AI Inputs Channel 4/Status/TxPDO State
//     PlcTask Inputs/GVL_iXlinker.EtherCAT_Master_EPPxxxx.Beckhoff_EPP3xxx.Beckhoff_EPP3xxxEK1122.A_0021_EPP3744_1041_0017.AI_Inputs_Channel_1.Status/TxPDO_Toggle <-> AI Inputs Channel 1/Status/TxPDO Toggle
//     PlcTask Inputs/GVL_iXlinker.EtherCAT_Master_EPPxxxx.Beckhoff_EPP3xxx.Beckhoff_EPP3xxxEK1122.A_0021_EPP3744_1041_0017.AI_Inputs_Channel_2.Status/TxPDO_Toggle <-> AI Inputs Channel 2/Status/TxPDO Toggle
//     PlcTask Inputs/GVL_iXlinker.EtherCAT_Master_EPPxxxx.Beckhoff_EPP3xxx.Beckhoff_EPP3xxxEK1122.A_0021_EPP3744_1041_0017.AI_Inputs_Channel_3.Status/TxPDO_Toggle <-> AI Inputs Channel 3/Status/TxPDO Toggle
//     PlcTask Inputs/GVL_iXlinker.EtherCAT_Master_EPPxxxx.Beckhoff_EPP3xxx.Beckhoff_EPP3xxxEK1122.A_0021_EPP3744_1041_0017.AI_Inputs_Channel_4.Status/TxPDO_Toggle <-> AI Inputs Channel 4/Status/TxPDO Toggle
//     PlcTask Inputs/GVL_iXlinker.EtherCAT_Master_EPPxxxx.Beckhoff_EPP3xxx.Beckhoff_EPP3xxxEK1122.A_0021_EPP3744_1041_0017.AI_Inputs_Channel_1.Value <-> AI Inputs Channel 1/Value
//     PlcTask Inputs/GVL_iXlinker.EtherCAT_Master_EPPxxxx.Beckhoff_EPP3xxx.Beckhoff_EPP3xxxEK1122.A_0021_EPP3744_1041_0017.AI_Inputs_Channel_2.Value <-> AI Inputs Channel 2/Value
//     PlcTask Inputs/GVL_iXlinker.EtherCAT_Master_EPPxxxx.Beckhoff_EPP3xxx.Beckhoff_EPP3xxxEK1122.A_0021_EPP3744_1041_0017.AI_Inputs_Channel_3.Value <-> AI Inputs Channel 3/Value
//     PlcTask Inputs/GVL_iXlinker.EtherCAT_Master_EPPxxxx.Beckhoff_EPP3xxx.Beckhoff_EPP3xxxEK1122.A_0021_EPP3744_1041_0017.AI_Inputs_Channel_4.Value <-> AI Inputs Channel 4/Value
//     PlcTask Inputs/GVL_iXlinker.EtherCAT_Master_EPPxxxx.Beckhoff_EPP3xxx.Beckhoff_EPP3xxxEK1122.A_0021_EPP3744_1041_0017.DEV_Inputs_Device.Safe_State_Active <-> DEV Inputs Device/Safe State Active
//     PlcTask Inputs/GVL_iXlinker.EtherCAT_Master_EPPxxxx.Beckhoff_EPP3xxx.Beckhoff_EPP3xxxEK1122.A_0021_EPP3744_1041_0017.DEV_Inputs_Device.Sync_error <-> DEV Inputs Device/Sync error
//     PlcTask Inputs/GVL_iXlinker.EtherCAT_Master_EPPxxxx.Beckhoff_EPP3xxx.Beckhoff_EPP3xxxEK1122.A_0021_EPP3744_1041_0017.DEV_Inputs_Device.Undervoltage_Us <-> DEV Inputs Device/Undervoltage Us
//     PlcTask Inputs/GVL_iXlinker.EtherCAT_Master_EPPxxxx.Beckhoff_EPP3xxx.Beckhoff_EPP3xxxEK1122.A_0021_EPP3744_1041_0017.DEV_Inputs_Device.Undervoltage_Up <-> DEV Inputs Device/Undervoltage Up
//     PlcTask Inputs/GVL_iXlinker.EtherCAT_Master_EPPxxxx.Beckhoff_EPP3xxx.Beckhoff_EPP3xxxEK1122.A_0021_EPP3744_1041_0017.DEV_Inputs_Device.TxPDO_Toggle <-> DEV Inputs Device/TxPDO Toggle
//     PlcTask Outputs/GVL_iXlinker.EtherCAT_Master_EPPxxxx.Beckhoff_EPP3xxx.Beckhoff_EPP3xxxEK1122.A_0021_EPP3744_1041_0017.DIG_Outputs.Output[0] <-> DIG Outputs/Output 1
//     PlcTask Outputs/GVL_iXlinker.EtherCAT_Master_EPPxxxx.Beckhoff_EPP3xxx.Beckhoff_EPP3xxxEK1122.A_0021_EPP3744_1041_0017.DIG_Outputs.Output[1] <-> DIG Outputs/Output 2
//     PlcTask Outputs/GVL_iXlinker.EtherCAT_Master_EPPxxxx.Beckhoff_EPP3xxx.Beckhoff_EPP3xxxEK1122.A_0021_EPP3744_1041_0017.DEV_Outputs_Device.Set_safe_state <-> DEV Outputs Device/Set safe state
//     PlcTask Inputs/GVL_iXlinker.EtherCAT_Master_EPPxxxx.Beckhoff_EPP3xxx.Beckhoff_EPP3xxxEK1122.A_0021_EPP3744_1041_0017.WcState.WcState <-> WcState/WcState
//     PlcTask Inputs/GVL_iXlinker.EtherCAT_Master_EPPxxxx.Beckhoff_EPP3xxx.Beckhoff_EPP3xxxEK1122.A_0021_EPP3744_1041_0017.WcState.InputToggle <-> WcState/InputToggle
//     PlcTask Inputs/GVL_iXlinker.EtherCAT_Master_EPPxxxx.Beckhoff_EPP3xxx.Beckhoff_EPP3xxxEK1122.A_0021_EPP3744_1041_0017.InfoData.AdsAddr <-> InfoData/AdsAddr
//     PlcTask Inputs/GVL_iXlinker.EtherCAT_Master_EPPxxxx.Beckhoff_EPP3xxx.Beckhoff_EPP3xxxEK1122.A_0021_EPP3744_1041_0017.InfoData.State <-> InfoData/State
//   PLC/PLC Instance <-> EtherCAT Master EPPxxxx/Beckhoff EPP3xxx/Beckhoff EPP3xxxEK1122/A_0022(EPP3744-1041-0018)
//     PlcTask Inputs/GVL_iXlinker.EtherCAT_Master_EPPxxxx.Beckhoff_EPP3xxx.Beckhoff_EPP3xxxEK1122.A_0022_EPP3744_1041_0018.DIG_Inputs.Input[0] <-> DIG Inputs/Input 1
//     PlcTask Inputs/GVL_iXlinker.EtherCAT_Master_EPPxxxx.Beckhoff_EPP3xxx.Beckhoff_EPP3xxxEK1122.A_0022_EPP3744_1041_0018.DIG_Inputs.Input[1] <-> DIG Inputs/Input 2
//     PlcTask Inputs/GVL_iXlinker.EtherCAT_Master_EPPxxxx.Beckhoff_EPP3xxx.Beckhoff_EPP3xxxEK1122.A_0022_EPP3744_1041_0018.DIG_Inputs.Input[2] <-> DIG Inputs/Input 3
//     PlcTask Inputs/GVL_iXlinker.EtherCAT_Master_EPPxxxx.Beckhoff_EPP3xxx.Beckhoff_EPP3xxxEK1122.A_0022_EPP3744_1041_0018.DIG_Inputs.Input[3] <-> DIG Inputs/Input 4
//     PlcTask Inputs/GVL_iXlinker.EtherCAT_Master_EPPxxxx.Beckhoff_EPP3xxx.Beckhoff_EPP3xxxEK1122.A_0022_EPP3744_1041_0018.DIG_Inputs.Input[4] <-> DIG Inputs/Input 5
//     PlcTask Inputs/GVL_iXlinker.EtherCAT_Master_EPPxxxx.Beckhoff_EPP3xxx.Beckhoff_EPP3xxxEK1122.A_0022_EPP3744_1041_0018.DIG_Inputs.Input[5] <-> DIG Inputs/Input 6
//     PlcTask Inputs/GVL_iXlinker.EtherCAT_Master_EPPxxxx.Beckhoff_EPP3xxx.Beckhoff_EPP3xxxEK1122.A_0022_EPP3744_1041_0018.AI_Inputs_Channel_1.Status/Underrange <-> AI Inputs Channel 1/Status/Underrange
//     PlcTask Inputs/GVL_iXlinker.EtherCAT_Master_EPPxxxx.Beckhoff_EPP3xxx.Beckhoff_EPP3xxxEK1122.A_0022_EPP3744_1041_0018.AI_Inputs_Channel_2.Status/Underrange <-> AI Inputs Channel 2/Status/Underrange
//     PlcTask Inputs/GVL_iXlinker.EtherCAT_Master_EPPxxxx.Beckhoff_EPP3xxx.Beckhoff_EPP3xxxEK1122.A_0022_EPP3744_1041_0018.AI_Inputs_Channel_3.Status/Underrange <-> AI Inputs Channel 3/Status/Underrange
//     PlcTask Inputs/GVL_iXlinker.EtherCAT_Master_EPPxxxx.Beckhoff_EPP3xxx.Beckhoff_EPP3xxxEK1122.A_0022_EPP3744_1041_0018.AI_Inputs_Channel_4.Status/Underrange <-> AI Inputs Channel 4/Status/Underrange
//     PlcTask Inputs/GVL_iXlinker.EtherCAT_Master_EPPxxxx.Beckhoff_EPP3xxx.Beckhoff_EPP3xxxEK1122.A_0022_EPP3744_1041_0018.AI_Inputs_Channel_1.Status/Overrange <-> AI Inputs Channel 1/Status/Overrange
//     PlcTask Inputs/GVL_iXlinker.EtherCAT_Master_EPPxxxx.Beckhoff_EPP3xxx.Beckhoff_EPP3xxxEK1122.A_0022_EPP3744_1041_0018.AI_Inputs_Channel_2.Status/Overrange <-> AI Inputs Channel 2/Status/Overrange
//     PlcTask Inputs/GVL_iXlinker.EtherCAT_Master_EPPxxxx.Beckhoff_EPP3xxx.Beckhoff_EPP3xxxEK1122.A_0022_EPP3744_1041_0018.AI_Inputs_Channel_3.Status/Overrange <-> AI Inputs Channel 3/Status/Overrange
//     PlcTask Inputs/GVL_iXlinker.EtherCAT_Master_EPPxxxx.Beckhoff_EPP3xxx.Beckhoff_EPP3xxxEK1122.A_0022_EPP3744_1041_0018.AI_Inputs_Channel_4.Status/Overrange <-> AI Inputs Channel 4/Status/Overrange
//     PlcTask Inputs/GVL_iXlinker.EtherCAT_Master_EPPxxxx.Beckhoff_EPP3xxx.Beckhoff_EPP3xxxEK1122.A_0022_EPP3744_1041_0018.AI_Inputs_Channel_1.Status/Limit_1 <-> AI Inputs Channel 1/Status/Limit 1
//     PlcTask Inputs/GVL_iXlinker.EtherCAT_Master_EPPxxxx.Beckhoff_EPP3xxx.Beckhoff_EPP3xxxEK1122.A_0022_EPP3744_1041_0018.AI_Inputs_Channel_1.Status/Limit_2 <-> AI Inputs Channel 1/Status/Limit 2
//     PlcTask Inputs/GVL_iXlinker.EtherCAT_Master_EPPxxxx.Beckhoff_EPP3xxx.Beckhoff_EPP3xxxEK1122.A_0022_EPP3744_1041_0018.AI_Inputs_Channel_2.Status/Limit_1 <-> AI Inputs Channel 2/Status/Limit 1
//     PlcTask Inputs/GVL_iXlinker.EtherCAT_Master_EPPxxxx.Beckhoff_EPP3xxx.Beckhoff_EPP3xxxEK1122.A_0022_EPP3744_1041_0018.AI_Inputs_Channel_2.Status/Limit_2 <-> AI Inputs Channel 2/Status/Limit 2
//     PlcTask Inputs/GVL_iXlinker.EtherCAT_Master_EPPxxxx.Beckhoff_EPP3xxx.Beckhoff_EPP3xxxEK1122.A_0022_EPP3744_1041_0018.AI_Inputs_Channel_3.Status/Limit_1 <-> AI Inputs Channel 3/Status/Limit 1
//     PlcTask Inputs/GVL_iXlinker.EtherCAT_Master_EPPxxxx.Beckhoff_EPP3xxx.Beckhoff_EPP3xxxEK1122.A_0022_EPP3744_1041_0018.AI_Inputs_Channel_3.Status/Limit_2 <-> AI Inputs Channel 3/Status/Limit 2
//     PlcTask Inputs/GVL_iXlinker.EtherCAT_Master_EPPxxxx.Beckhoff_EPP3xxx.Beckhoff_EPP3xxxEK1122.A_0022_EPP3744_1041_0018.AI_Inputs_Channel_4.Status/Limit_1 <-> AI Inputs Channel 4/Status/Limit 1
//     PlcTask Inputs/GVL_iXlinker.EtherCAT_Master_EPPxxxx.Beckhoff_EPP3xxx.Beckhoff_EPP3xxxEK1122.A_0022_EPP3744_1041_0018.AI_Inputs_Channel_4.Status/Limit_2 <-> AI Inputs Channel 4/Status/Limit 2
//     PlcTask Inputs/GVL_iXlinker.EtherCAT_Master_EPPxxxx.Beckhoff_EPP3xxx.Beckhoff_EPP3xxxEK1122.A_0022_EPP3744_1041_0018.AI_Inputs_Channel_1.Status/Error <-> AI Inputs Channel 1/Status/Error
//     PlcTask Inputs/GVL_iXlinker.EtherCAT_Master_EPPxxxx.Beckhoff_EPP3xxx.Beckhoff_EPP3xxxEK1122.A_0022_EPP3744_1041_0018.AI_Inputs_Channel_2.Status/Error <-> AI Inputs Channel 2/Status/Error
//     PlcTask Inputs/GVL_iXlinker.EtherCAT_Master_EPPxxxx.Beckhoff_EPP3xxx.Beckhoff_EPP3xxxEK1122.A_0022_EPP3744_1041_0018.AI_Inputs_Channel_3.Status/Error <-> AI Inputs Channel 3/Status/Error
//     PlcTask Inputs/GVL_iXlinker.EtherCAT_Master_EPPxxxx.Beckhoff_EPP3xxx.Beckhoff_EPP3xxxEK1122.A_0022_EPP3744_1041_0018.AI_Inputs_Channel_4.Status/Error <-> AI Inputs Channel 4/Status/Error
//     PlcTask Inputs/GVL_iXlinker.EtherCAT_Master_EPPxxxx.Beckhoff_EPP3xxx.Beckhoff_EPP3xxxEK1122.A_0022_EPP3744_1041_0018.AI_Inputs_Channel_1.Status/TxPDO_State <-> AI Inputs Channel 1/Status/TxPDO State
//     PlcTask Inputs/GVL_iXlinker.EtherCAT_Master_EPPxxxx.Beckhoff_EPP3xxx.Beckhoff_EPP3xxxEK1122.A_0022_EPP3744_1041_0018.AI_Inputs_Channel_2.Status/TxPDO_State <-> AI Inputs Channel 2/Status/TxPDO State
//     PlcTask Inputs/GVL_iXlinker.EtherCAT_Master_EPPxxxx.Beckhoff_EPP3xxx.Beckhoff_EPP3xxxEK1122.A_0022_EPP3744_1041_0018.AI_Inputs_Channel_3.Status/TxPDO_State <-> AI Inputs Channel 3/Status/TxPDO State
//     PlcTask Inputs/GVL_iXlinker.EtherCAT_Master_EPPxxxx.Beckhoff_EPP3xxx.Beckhoff_EPP3xxxEK1122.A_0022_EPP3744_1041_0018.AI_Inputs_Channel_4.Status/TxPDO_State <-> AI Inputs Channel 4/Status/TxPDO State
//     PlcTask Inputs/GVL_iXlinker.EtherCAT_Master_EPPxxxx.Beckhoff_EPP3xxx.Beckhoff_EPP3xxxEK1122.A_0022_EPP3744_1041_0018.AI_Inputs_Channel_1.Status/TxPDO_Toggle <-> AI Inputs Channel 1/Status/TxPDO Toggle
//     PlcTask Inputs/GVL_iXlinker.EtherCAT_Master_EPPxxxx.Beckhoff_EPP3xxx.Beckhoff_EPP3xxxEK1122.A_0022_EPP3744_1041_0018.AI_Inputs_Channel_2.Status/TxPDO_Toggle <-> AI Inputs Channel 2/Status/TxPDO Toggle
//     PlcTask Inputs/GVL_iXlinker.EtherCAT_Master_EPPxxxx.Beckhoff_EPP3xxx.Beckhoff_EPP3xxxEK1122.A_0022_EPP3744_1041_0018.AI_Inputs_Channel_3.Status/TxPDO_Toggle <-> AI Inputs Channel 3/Status/TxPDO Toggle
//     PlcTask Inputs/GVL_iXlinker.EtherCAT_Master_EPPxxxx.Beckhoff_EPP3xxx.Beckhoff_EPP3xxxEK1122.A_0022_EPP3744_1041_0018.AI_Inputs_Channel_4.Status/TxPDO_Toggle <-> AI Inputs Channel 4/Status/TxPDO Toggle
//     PlcTask Inputs/GVL_iXlinker.EtherCAT_Master_EPPxxxx.Beckhoff_EPP3xxx.Beckhoff_EPP3xxxEK1122.A_0022_EPP3744_1041_0018.AI_Inputs_Channel_1.Value <-> AI Inputs Channel 1/Value
//     PlcTask Inputs/GVL_iXlinker.EtherCAT_Master_EPPxxxx.Beckhoff_EPP3xxx.Beckhoff_EPP3xxxEK1122.A_0022_EPP3744_1041_0018.AI_Inputs_Channel_2.Value <-> AI Inputs Channel 2/Value
//     PlcTask Inputs/GVL_iXlinker.EtherCAT_Master_EPPxxxx.Beckhoff_EPP3xxx.Beckhoff_EPP3xxxEK1122.A_0022_EPP3744_1041_0018.AI_Inputs_Channel_3.Value <-> AI Inputs Channel 3/Value
//     PlcTask Inputs/GVL_iXlinker.EtherCAT_Master_EPPxxxx.Beckhoff_EPP3xxx.Beckhoff_EPP3xxxEK1122.A_0022_EPP3744_1041_0018.AI_Inputs_Channel_4.Value <-> AI Inputs Channel 4/Value
//     PlcTask Inputs/GVL_iXlinker.EtherCAT_Master_EPPxxxx.Beckhoff_EPP3xxx.Beckhoff_EPP3xxxEK1122.A_0022_EPP3744_1041_0018.DEV_Inputs_Device.Safe_State_Active <-> DEV Inputs Device/Safe State Active
//     PlcTask Inputs/GVL_iXlinker.EtherCAT_Master_EPPxxxx.Beckhoff_EPP3xxx.Beckhoff_EPP3xxxEK1122.A_0022_EPP3744_1041_0018.DEV_Inputs_Device.Sync_error <-> DEV Inputs Device/Sync error
//     PlcTask Inputs/GVL_iXlinker.EtherCAT_Master_EPPxxxx.Beckhoff_EPP3xxx.Beckhoff_EPP3xxxEK1122.A_0022_EPP3744_1041_0018.DEV_Inputs_Device.Undervoltage_Us <-> DEV Inputs Device/Undervoltage Us
//     PlcTask Inputs/GVL_iXlinker.EtherCAT_Master_EPPxxxx.Beckhoff_EPP3xxx.Beckhoff_EPP3xxxEK1122.A_0022_EPP3744_1041_0018.DEV_Inputs_Device.Undervoltage_Up <-> DEV Inputs Device/Undervoltage Up
//     PlcTask Inputs/GVL_iXlinker.EtherCAT_Master_EPPxxxx.Beckhoff_EPP3xxx.Beckhoff_EPP3xxxEK1122.A_0022_EPP3744_1041_0018.DEV_Inputs_Device.TxPDO_Toggle <-> DEV Inputs Device/TxPDO Toggle
//     PlcTask Outputs/GVL_iXlinker.EtherCAT_Master_EPPxxxx.Beckhoff_EPP3xxx.Beckhoff_EPP3xxxEK1122.A_0022_EPP3744_1041_0018.DIG_Outputs.Output[0] <-> DIG Outputs/Output 1
//     PlcTask Outputs/GVL_iXlinker.EtherCAT_Master_EPPxxxx.Beckhoff_EPP3xxx.Beckhoff_EPP3xxxEK1122.A_0022_EPP3744_1041_0018.DIG_Outputs.Output[1] <-> DIG Outputs/Output 2
//     PlcTask Outputs/GVL_iXlinker.EtherCAT_Master_EPPxxxx.Beckhoff_EPP3xxx.Beckhoff_EPP3xxxEK1122.A_0022_EPP3744_1041_0018.DEV_Outputs_Device.Set_safe_state <-> DEV Outputs Device/Set safe state
//     PlcTask Inputs/GVL_iXlinker.EtherCAT_Master_EPPxxxx.Beckhoff_EPP3xxx.Beckhoff_EPP3xxxEK1122.A_0022_EPP3744_1041_0018.WcState.WcState <-> WcState/WcState
//     PlcTask Inputs/GVL_iXlinker.EtherCAT_Master_EPPxxxx.Beckhoff_EPP3xxx.Beckhoff_EPP3xxxEK1122.A_0022_EPP3744_1041_0018.WcState.InputToggle <-> WcState/InputToggle
//     PlcTask Inputs/GVL_iXlinker.EtherCAT_Master_EPPxxxx.Beckhoff_EPP3xxx.Beckhoff_EPP3xxxEK1122.A_0022_EPP3744_1041_0018.InfoData.AdsAddr <-> InfoData/AdsAddr
//     PlcTask Inputs/GVL_iXlinker.EtherCAT_Master_EPPxxxx.Beckhoff_EPP3xxx.Beckhoff_EPP3xxxEK1122.A_0022_EPP3744_1041_0018.InfoData.State <-> InfoData/State
//   PLC/PLC Instance <-> EtherCAT Master EPPxxxx/Beckhoff EPP3xxx/Beckhoff EPP3xxxEK1122/A_0023(EPP3744-1041-0019)
//     PlcTask Inputs/GVL_iXlinker.EtherCAT_Master_EPPxxxx.Beckhoff_EPP3xxx.Beckhoff_EPP3xxxEK1122.A_0023_EPP3744_1041_0019.DIG_Inputs.Input[0] <-> DIG Inputs/Input 1
//     PlcTask Inputs/GVL_iXlinker.EtherCAT_Master_EPPxxxx.Beckhoff_EPP3xxx.Beckhoff_EPP3xxxEK1122.A_0023_EPP3744_1041_0019.DIG_Inputs.Input[1] <-> DIG Inputs/Input 2
//     PlcTask Inputs/GVL_iXlinker.EtherCAT_Master_EPPxxxx.Beckhoff_EPP3xxx.Beckhoff_EPP3xxxEK1122.A_0023_EPP3744_1041_0019.DIG_Inputs.Input[2] <-> DIG Inputs/Input 3
//     PlcTask Inputs/GVL_iXlinker.EtherCAT_Master_EPPxxxx.Beckhoff_EPP3xxx.Beckhoff_EPP3xxxEK1122.A_0023_EPP3744_1041_0019.DIG_Inputs.Input[3] <-> DIG Inputs/Input 4
//     PlcTask Inputs/GVL_iXlinker.EtherCAT_Master_EPPxxxx.Beckhoff_EPP3xxx.Beckhoff_EPP3xxxEK1122.A_0023_EPP3744_1041_0019.DIG_Inputs.Input[4] <-> DIG Inputs/Input 5
//     PlcTask Inputs/GVL_iXlinker.EtherCAT_Master_EPPxxxx.Beckhoff_EPP3xxx.Beckhoff_EPP3xxxEK1122.A_0023_EPP3744_1041_0019.DIG_Inputs.Input[5] <-> DIG Inputs/Input 6
//     PlcTask Inputs/GVL_iXlinker.EtherCAT_Master_EPPxxxx.Beckhoff_EPP3xxx.Beckhoff_EPP3xxxEK1122.A_0023_EPP3744_1041_0019.AI_Inputs_Channel_1.Status/Underrange <-> AI Inputs Channel 1/Status/Underrange
//     PlcTask Inputs/GVL_iXlinker.EtherCAT_Master_EPPxxxx.Beckhoff_EPP3xxx.Beckhoff_EPP3xxxEK1122.A_0023_EPP3744_1041_0019.AI_Inputs_Channel_2.Status/Underrange <-> AI Inputs Channel 2/Status/Underrange
//     PlcTask Inputs/GVL_iXlinker.EtherCAT_Master_EPPxxxx.Beckhoff_EPP3xxx.Beckhoff_EPP3xxxEK1122.A_0023_EPP3744_1041_0019.AI_Inputs_Channel_3.Status/Underrange <-> AI Inputs Channel 3/Status/Underrange
//     PlcTask Inputs/GVL_iXlinker.EtherCAT_Master_EPPxxxx.Beckhoff_EPP3xxx.Beckhoff_EPP3xxxEK1122.A_0023_EPP3744_1041_0019.AI_Inputs_Channel_4.Status/Underrange <-> AI Inputs Channel 4/Status/Underrange
//     PlcTask Inputs/GVL_iXlinker.EtherCAT_Master_EPPxxxx.Beckhoff_EPP3xxx.Beckhoff_EPP3xxxEK1122.A_0023_EPP3744_1041_0019.AI_Inputs_Channel_1.Status/Overrange <-> AI Inputs Channel 1/Status/Overrange
//     PlcTask Inputs/GVL_iXlinker.EtherCAT_Master_EPPxxxx.Beckhoff_EPP3xxx.Beckhoff_EPP3xxxEK1122.A_0023_EPP3744_1041_0019.AI_Inputs_Channel_2.Status/Overrange <-> AI Inputs Channel 2/Status/Overrange
//     PlcTask Inputs/GVL_iXlinker.EtherCAT_Master_EPPxxxx.Beckhoff_EPP3xxx.Beckhoff_EPP3xxxEK1122.A_0023_EPP3744_1041_0019.AI_Inputs_Channel_3.Status/Overrange <-> AI Inputs Channel 3/Status/Overrange
//     PlcTask Inputs/GVL_iXlinker.EtherCAT_Master_EPPxxxx.Beckhoff_EPP3xxx.Beckhoff_EPP3xxxEK1122.A_0023_EPP3744_1041_0019.AI_Inputs_Channel_4.Status/Overrange <-> AI Inputs Channel 4/Status/Overrange
//     PlcTask Inputs/GVL_iXlinker.EtherCAT_Master_EPPxxxx.Beckhoff_EPP3xxx.Beckhoff_EPP3xxxEK1122.A_0023_EPP3744_1041_0019.AI_Inputs_Channel_1.Status/Limit_1 <-> AI Inputs Channel 1/Status/Limit 1
//     PlcTask Inputs/GVL_iXlinker.EtherCAT_Master_EPPxxxx.Beckhoff_EPP3xxx.Beckhoff_EPP3xxxEK1122.A_0023_EPP3744_1041_0019.AI_Inputs_Channel_1.Status/Limit_2 <-> AI Inputs Channel 1/Status/Limit 2
//     PlcTask Inputs/GVL_iXlinker.EtherCAT_Master_EPPxxxx.Beckhoff_EPP3xxx.Beckhoff_EPP3xxxEK1122.A_0023_EPP3744_1041_0019.AI_Inputs_Channel_2.Status/Limit_1 <-> AI Inputs Channel 2/Status/Limit 1
//     PlcTask Inputs/GVL_iXlinker.EtherCAT_Master_EPPxxxx.Beckhoff_EPP3xxx.Beckhoff_EPP3xxxEK1122.A_0023_EPP3744_1041_0019.AI_Inputs_Channel_2.Status/Limit_2 <-> AI Inputs Channel 2/Status/Limit 2
//     PlcTask Inputs/GVL_iXlinker.EtherCAT_Master_EPPxxxx.Beckhoff_EPP3xxx.Beckhoff_EPP3xxxEK1122.A_0023_EPP3744_1041_0019.AI_Inputs_Channel_3.Status/Limit_1 <-> AI Inputs Channel 3/Status/Limit 1
//     PlcTask Inputs/GVL_iXlinker.EtherCAT_Master_EPPxxxx.Beckhoff_EPP3xxx.Beckhoff_EPP3xxxEK1122.A_0023_EPP3744_1041_0019.AI_Inputs_Channel_3.Status/Limit_2 <-> AI Inputs Channel 3/Status/Limit 2
//     PlcTask Inputs/GVL_iXlinker.EtherCAT_Master_EPPxxxx.Beckhoff_EPP3xxx.Beckhoff_EPP3xxxEK1122.A_0023_EPP3744_1041_0019.AI_Inputs_Channel_4.Status/Limit_1 <-> AI Inputs Channel 4/Status/Limit 1
//     PlcTask Inputs/GVL_iXlinker.EtherCAT_Master_EPPxxxx.Beckhoff_EPP3xxx.Beckhoff_EPP3xxxEK1122.A_0023_EPP3744_1041_0019.AI_Inputs_Channel_4.Status/Limit_2 <-> AI Inputs Channel 4/Status/Limit 2
//     PlcTask Inputs/GVL_iXlinker.EtherCAT_Master_EPPxxxx.Beckhoff_EPP3xxx.Beckhoff_EPP3xxxEK1122.A_0023_EPP3744_1041_0019.AI_Inputs_Channel_1.Status/Error <-> AI Inputs Channel 1/Status/Error
//     PlcTask Inputs/GVL_iXlinker.EtherCAT_Master_EPPxxxx.Beckhoff_EPP3xxx.Beckhoff_EPP3xxxEK1122.A_0023_EPP3744_1041_0019.AI_Inputs_Channel_2.Status/Error <-> AI Inputs Channel 2/Status/Error
//     PlcTask Inputs/GVL_iXlinker.EtherCAT_Master_EPPxxxx.Beckhoff_EPP3xxx.Beckhoff_EPP3xxxEK1122.A_0023_EPP3744_1041_0019.AI_Inputs_Channel_3.Status/Error <-> AI Inputs Channel 3/Status/Error
//     PlcTask Inputs/GVL_iXlinker.EtherCAT_Master_EPPxxxx.Beckhoff_EPP3xxx.Beckhoff_EPP3xxxEK1122.A_0023_EPP3744_1041_0019.AI_Inputs_Channel_4.Status/Error <-> AI Inputs Channel 4/Status/Error
//     PlcTask Inputs/GVL_iXlinker.EtherCAT_Master_EPPxxxx.Beckhoff_EPP3xxx.Beckhoff_EPP3xxxEK1122.A_0023_EPP3744_1041_0019.AI_Inputs_Channel_1.Status/TxPDO_State <-> AI Inputs Channel 1/Status/TxPDO State
//     PlcTask Inputs/GVL_iXlinker.EtherCAT_Master_EPPxxxx.Beckhoff_EPP3xxx.Beckhoff_EPP3xxxEK1122.A_0023_EPP3744_1041_0019.AI_Inputs_Channel_2.Status/TxPDO_State <-> AI Inputs Channel 2/Status/TxPDO State
//     PlcTask Inputs/GVL_iXlinker.EtherCAT_Master_EPPxxxx.Beckhoff_EPP3xxx.Beckhoff_EPP3xxxEK1122.A_0023_EPP3744_1041_0019.AI_Inputs_Channel_3.Status/TxPDO_State <-> AI Inputs Channel 3/Status/TxPDO State
//     PlcTask Inputs/GVL_iXlinker.EtherCAT_Master_EPPxxxx.Beckhoff_EPP3xxx.Beckhoff_EPP3xxxEK1122.A_0023_EPP3744_1041_0019.AI_Inputs_Channel_4.Status/TxPDO_State <-> AI Inputs Channel 4/Status/TxPDO State
//     PlcTask Inputs/GVL_iXlinker.EtherCAT_Master_EPPxxxx.Beckhoff_EPP3xxx.Beckhoff_EPP3xxxEK1122.A_0023_EPP3744_1041_0019.AI_Inputs_Channel_1.Status/TxPDO_Toggle <-> AI Inputs Channel 1/Status/TxPDO Toggle
//     PlcTask Inputs/GVL_iXlinker.EtherCAT_Master_EPPxxxx.Beckhoff_EPP3xxx.Beckhoff_EPP3xxxEK1122.A_0023_EPP3744_1041_0019.AI_Inputs_Channel_2.Status/TxPDO_Toggle <-> AI Inputs Channel 2/Status/TxPDO Toggle
//     PlcTask Inputs/GVL_iXlinker.EtherCAT_Master_EPPxxxx.Beckhoff_EPP3xxx.Beckhoff_EPP3xxxEK1122.A_0023_EPP3744_1041_0019.AI_Inputs_Channel_3.Status/TxPDO_Toggle <-> AI Inputs Channel 3/Status/TxPDO Toggle
//     PlcTask Inputs/GVL_iXlinker.EtherCAT_Master_EPPxxxx.Beckhoff_EPP3xxx.Beckhoff_EPP3xxxEK1122.A_0023_EPP3744_1041_0019.AI_Inputs_Channel_4.Status/TxPDO_Toggle <-> AI Inputs Channel 4/Status/TxPDO Toggle
//     PlcTask Inputs/GVL_iXlinker.EtherCAT_Master_EPPxxxx.Beckhoff_EPP3xxx.Beckhoff_EPP3xxxEK1122.A_0023_EPP3744_1041_0019.AI_Inputs_Channel_1.Value <-> AI Inputs Channel 1/Value
